// TwinCAT 3 PLC project sample_delivery
// Title: lcsl-plc-icl-sample-delivery
// Company: SLAC
// ProjectVersion: 0.0.0
// ProgramVersion: 3.1.4023.0
// libraries:
//   lcls-twincat-sample-delivery, * (SLAC)
//   Tc2_Standard, * (Beckhoff Automation GmbH)
//   Tc2_System, * (Beckhoff Automation GmbH)
//   Tc3_Module, * (Beckhoff Automation GmbH)
// project tree:
//   GVLs/ GVL_SDS.TcGVL
//   / PlcTask.TcTTO (not stored), SerialComm.TcTTO (not stored)
//   POUs/ MAIN.TcPOU, SerialTxRx.TcPOU (not stored)
// real-time tasks:
//   TASK PlcTask: cycle T#10ms, priority 20, ADS port 351
//   TASK SerialComm: cycle T#5ms, priority 1, ADS port 350
// I/O:
//   DEVICE MAIN (EtherCAT), AmsNetId 0.0.0.0.2.1
//     Term 65 (EK1200) [EK1200-5000 EtherCAT Power supply (2A E-Bus)]
//       Term 66 (EL6070) [EL6070 1Ch. Licensing-Terminal]
//       Term 67 (EK1110) [EK1110 EtherCAT extension]
//     Box 68 (EP9128-0021) [EP9128-0021 8x EtherCAT junction]
//       Term 69 (EP9128-1021) [EP9128-1021 8x EtherCAT junction - Dev A]
//       Term 70 (EP9128-2021) [EP9128-2021 8x EtherCAT junction - Dev B]
//     Box 23 (EP9128-0021) [EP9128-0021 8x EtherCAT junction]
//       Term 71 (EP9128-1021) [EP9128-1021 8x EtherCAT junction - Dev A]
//       Term 72 (EP9128-2021) [EP9128-2021 8x EtherCAT junction - Dev B]
//     ALI (EP1111) [EP1111-0000 ID-Switch]
//     ALI_X (EP7041-0002) [EP7041-0002 1Ch. Stepper motor output stage (50V, 5A)]
//     ALI_Y (EP7041-0002) [EP7041-0002 1Ch. Stepper motor output stage (50V, 5A)]
//     ALI_Z (EP7041-0002) [EP7041-0002 1Ch. Stepper motor output stage (50V, 5A)]
//     ALI_X_ENC (EP5101-0011) [EP5101-0011 1Ch. Inc. Encoder 5V, D-SUB15]
//     ALI_Gauges (EP3174-0002) [EP3174-0002 4Ch. Ana. Input +/-10V, 0-10V, 0/4-20mA configurable]
//     ALI_PropValve (EP7041-0002) [EP7041-0002 1Ch. Stepper motor output stage (50V, 5A)]
//     ALI_Y_ENC (EP5101-0011) [EP5101-0011 1Ch. Inc. Encoder 5V, D-SUB15]
//     ALI_DIO (EP2338-0001) [EP2338-0001 8 Ch. Dig. Input/Output 24V, 0,5A, M8]
//     M3 Selector A (EP1111) [EP1111-0000 ID-Switch]
//     M3 Selector A Digital IO (EP2338-1001) [EP2338-1001 8 Ch. Dig. Input/Output 24V, 3ms, 0,5A, M8]
//     M3 Selector A Serial IO (EP6002-0002) [EP6002-0002 Interface (RS232/422/485)]
//     M3 Selector B (EP1111) [EP1111-0000 ID-Switch]
//     M3 Selector B Digital IO (EP2338-1001) [EP2338-1001 8 Ch. Dig. Input/Output 24V, 3ms, 0,5A, M8]
//     M3 Selector B Serial IO (EP6002-0002) [EP6002-0002 Interface (RS232/422/485)]
//     PCM A (EP1111) [EP1111-0000 ID-Switch]
//     PCM A (EP4374-0002) [EP4374-0002 2Ch. Ana. Input +/-10V, 0-10V, 0/4-20mA configurable; 2Ch. Ana. Output +/-10V, 0-10V, 0/4-20mA configurable]
//     PCM A (EP3174-0002) [EP3174-0002 4Ch. Ana. Input +/-10V, 0-10V, 0/4-20mA configurable]
//     PCM A (EP6002-0002) [EP6002-0002 Interface (RS232/422/485)]
//     PCM B (EP1111) [EP1111-0000 ID-Switch]
//     PCM B (EP4374-0002) [EP4374-0002 2Ch. Ana. Input +/-10V, 0-10V, 0/4-20mA configurable; 2Ch. Ana. Output +/-10V, 0-10V, 0/4-20mA configurable]
//     PCM B (EP3174-0002) [EP3174-0002 4Ch. Ana. Input +/-10V, 0-10V, 0/4-20mA configurable]
//     PCM B (EP6002-0002) [EP6002-0002 Interface (RS232/422/485)]
//     Gas_Mani (EP1111) [EP1111-0000 ID-Switch]
//     Gas_Mani_NeedleValve (EP4374-0002) [EP4374-0002 2Ch. Ana. Input +/-10V, 0-10V, 0/4-20mA configurable; 2Ch. Ana. Output +/-10V, 0-10V, 0/4-20mA configurable]
//     Gas_Mani_ValveCtrl (EP2338-0001) [EP2338-0001 8 Ch. Dig. Input/Output 24V, 0,5A, M8]
//     Gas_Mani_ValveRbk (EP2338-0001) [EP2338-0001 8 Ch. Dig. Input/Output 24V, 0,5A, M8]
//     M3 Selector C (EP1111) [EP1111-0000 ID-Switch]
//     M3 Selector C Digital IO (EP2338-1001) [EP2338-1001 8 Ch. Dig. Input/Output 24V, 3ms, 0,5A, M8]
//     M3 Selector C Serial IO (EP6002-0002) [EP6002-0002 Interface (RS232/422/485)]
//     M3 Selector D (EP1111) [EP1111-0000 ID-Switch]
//     M3 Selector D Digital IO (EP2338-1001) [EP2338-1001 8 Ch. Dig. Input/Output 24V, 3ms, 0,5A, M8]
//     M3 Selector D Serial IO (EP6002-0002) [EP6002-0002 Interface (RS232/422/485)]
//     PCM C (EP1111) [EP1111-0000 ID-Switch]
//     PCM C (EP4374-0002) [EP4374-0002 2Ch. Ana. Input +/-10V, 0-10V, 0/4-20mA configurable; 2Ch. Ana. Output +/-10V, 0-10V, 0/4-20mA configurable]
//     PCM C (EP3174-0002) [EP3174-0002 4Ch. Ana. Input +/-10V, 0-10V, 0/4-20mA configurable]
//     PCM C (EP6002-0002) [EP6002-0002 Interface (RS232/422/485)]
//     PCM D (EP1111) [EP1111-0000 ID-Switch]
//     PCM D (EP4374-0002) [EP4374-0002 2Ch. Ana. Input +/-10V, 0-10V, 0/4-20mA configurable; 2Ch. Ana. Output +/-10V, 0-10V, 0/4-20mA configurable]
//     PCM D (EP3174-0002) [EP3174-0002 4Ch. Ana. Input +/-10V, 0-10V, 0/4-20mA configurable]
//     PCM D (EP6002-0002) [EP6002-0002 Interface (RS232/422/485)]
//     Bronkhorst MFM A [Mass Flow / Pressure Controller - Slave]
//     Bronkhorst MFM B [Mass Flow / Pressure Controller - Slave]
//     Bronkhorst MFM C [Mass Flow / Pressure Controller - Slave]
//     Bronkhorst MFM D [Mass Flow / Pressure Controller - Slave]
//     Solenoid Pair A (EP1111)
//     Solenoid Pair A Digital IO (EP2338-0001)
//     SC5 [EP9128-0021 8x EtherCAT junction]
//       Box 26 (EP9128-1021) [EP9128-1021 8x EtherCAT junction - Dev A]
//       Box 27 (EP9128-2021) [EP9128-2021 8x EtherCAT junction - Dev B]
//     SC4 [EP9128-0021 8x EtherCAT junction]
//       Box 24 (EP9128-1021) [EP9128-1021 8x EtherCAT junction - Dev A]
//       Box 25 (EP9128-2021) [EP9128-2021 8x EtherCAT junction - Dev B]
// variable links:
//   sample_delivery Instance <-> MAIN (EtherCAT)/Bronkhorst MFM A
//     PlcTask Inputs/GVL_SDS.BronkhorstA.stMFM.i_rFlow <-> TxPDO Map/fMeasure
//     PlcTask Outputs/GVL_SDS.BronkhorstA.stMFM.q_rSetpoint <-> RxPDO Map/fSetpoint
//   sample_delivery Instance <-> MAIN (EtherCAT)/Bronkhorst MFM B
//     PlcTask Inputs/GVL_SDS.BronkhorstB.stMFM.i_rFlow <-> TxPDO Map/fMeasure
//     PlcTask Outputs/GVL_SDS.BronkhorstB.stMFM.q_rSetpoint <-> RxPDO Map/fSetpoint
//   sample_delivery Instance <-> MAIN (EtherCAT)/Bronkhorst MFM C
//     PlcTask Inputs/GVL_SDS.BronkhorstC.stMFM.i_rFlow <-> TxPDO Map/fMeasure
//     PlcTask Outputs/GVL_SDS.BronkhorstC.stMFM.q_rSetpoint <-> RxPDO Map/fSetpoint
//   sample_delivery Instance <-> MAIN (EtherCAT)/Bronkhorst MFM D
//     PlcTask Inputs/GVL_SDS.BronkhorstD.stMFM.i_rFlow <-> TxPDO Map/fMeasure
//     PlcTask Outputs/GVL_SDS.BronkhorstD.stMFM.q_rSetpoint <-> RxPDO Map/fSetpoint
//   sample_delivery Instance <-> MAIN (EtherCAT)/Gas_Mani (EP1111)
//     PlcTask Inputs/GVL_SDS.GasMan.stBaseIO.i_SyncUnitWC <-> WcState/WcState
//   sample_delivery Instance <-> MAIN (EtherCAT)/Gas_Mani_ValveCtrl (EP2338-0001)
//     PlcTask Outputs/GVL_SDS.GasMan.stValve[{1..7}].qxDO <-> Channel {9..15}/Output  (7 links)
//   sample_delivery Instance <-> MAIN (EtherCAT)/Gas_Mani_ValveRbk (EP2338-0001)
//     PlcTask Inputs/GVL_SDS.GasMan.stValve[{1..7}].ixOPN <-> Channel {1..7}/Input  (7 links)
//   sample_delivery Instance <-> MAIN (EtherCAT)/M3 Selector A (EP1111)
//     PlcTask Inputs/GVL_SDS.M3SelectorA.stBaseIO.i_SyncUnitWC <-> WcState/WcState
//   sample_delivery Instance <-> MAIN (EtherCAT)/M3 Selector A Digital IO (EP2338-1001)
//     PlcTask Outputs/GVL_SDS.M3SelectorA.stShaker01.q_xPwrDO <-> Channel 9/Output
//     PlcTask Outputs/GVL_SDS.M3SelectorA.stShaker02.q_xPwrDO <-> Channel 10/Output
//     PlcTask Outputs/GVL_SDS.M3SelectorA.stShaker03.q_xPwrDO <-> Channel 11/Output
//     PlcTask Outputs/GVL_SDS.M3SelectorA.stShaker04.q_xPwrDO <-> Channel 12/Output
//   sample_delivery Instance <-> MAIN (EtherCAT)/M3 Selector A Serial IO (EP6002-0002)
//     SerialComm Inputs/GVL_SDS.M3SelectorA.stSensSerial.stComIn/D <-> COM TxPDO-Map Inputs Channel 1/Data In 0
//     SerialComm Inputs/GVL_SDS.M3SelectorA.stSensSerial.stComIn/D @bit {8..168 step 8} <-> COM TxPDO-Map Inputs Channel 1/Data In {1..21}  (21 links)
//     SerialComm Inputs/GVL_SDS.M3SelectorA.stSensSerial.stComIn/Status <-> COM TxPDO-Map Inputs Channel 1/Status
//     SerialComm Inputs/GVL_SDS.M3SelectorA.stViciSerial.stComIn/D <-> COM TxPDO-Map Inputs Channel 2/Data In 0
//     SerialComm Inputs/GVL_SDS.M3SelectorA.stViciSerial.stComIn/D @bit {8..168 step 8} <-> COM TxPDO-Map Inputs Channel 2/Data In {1..21}  (21 links)
//     SerialComm Inputs/GVL_SDS.M3SelectorA.stViciSerial.stComIn/Status <-> COM TxPDO-Map Inputs Channel 2/Status
//     SerialComm Outputs/GVL_SDS.M3SelectorA.stSensSerial.stComOut/Ctrl <-> COM RxPDO-Map Outputs Channel 1/Ctrl
//     SerialComm Outputs/GVL_SDS.M3SelectorA.stSensSerial.stComOut/D <-> COM RxPDO-Map Outputs Channel 1/Data Out 0
//     SerialComm Outputs/GVL_SDS.M3SelectorA.stSensSerial.stComOut/D @bit {8..168 step 8} <-> COM RxPDO-Map Outputs Channel 1/Data Out {1..21}  (21 links)
//     SerialComm Outputs/GVL_SDS.M3SelectorA.stViciSerial.stComOut/Ctrl <-> COM RxPDO-Map Outputs Channel 2/Ctrl
//     SerialComm Outputs/GVL_SDS.M3SelectorA.stViciSerial.stComOut/D <-> COM RxPDO-Map Outputs Channel 2/Data Out 0
//     SerialComm Outputs/GVL_SDS.M3SelectorA.stViciSerial.stComOut/D @bit {8..168 step 8} <-> COM RxPDO-Map Outputs Channel 2/Data Out {1..21}  (21 links)
//   sample_delivery Instance <-> MAIN (EtherCAT)/M3 Selector B (EP1111)
//     PlcTask Inputs/GVL_SDS.M3SelectorB.stBaseIO.i_SyncUnitWC <-> WcState/WcState
//   sample_delivery Instance <-> MAIN (EtherCAT)/M3 Selector B Digital IO (EP2338-1001)
//     PlcTask Outputs/GVL_SDS.M3SelectorB.stShaker01.q_xPwrDO <-> Channel 9/Output
//     PlcTask Outputs/GVL_SDS.M3SelectorB.stShaker02.q_xPwrDO <-> Channel 10/Output
//     PlcTask Outputs/GVL_SDS.M3SelectorB.stShaker03.q_xPwrDO <-> Channel 11/Output
//     PlcTask Outputs/GVL_SDS.M3SelectorB.stShaker04.q_xPwrDO <-> Channel 12/Output
//   sample_delivery Instance <-> MAIN (EtherCAT)/M3 Selector B Serial IO (EP6002-0002)
//     SerialComm Inputs/GVL_SDS.M3SelectorB.stSensSerial.stComIn/D <-> COM TxPDO-Map Inputs Channel 1/Data In 0
//     SerialComm Inputs/GVL_SDS.M3SelectorB.stSensSerial.stComIn/D @bit {8..168 step 8} <-> COM TxPDO-Map Inputs Channel 1/Data In {1..21}  (21 links)
//     SerialComm Inputs/GVL_SDS.M3SelectorB.stSensSerial.stComIn/Status <-> COM TxPDO-Map Inputs Channel 1/Status
//     SerialComm Inputs/GVL_SDS.M3SelectorB.stViciSerial.stComIn/D <-> COM TxPDO-Map Inputs Channel 2/Data In 0
//     SerialComm Inputs/GVL_SDS.M3SelectorB.stViciSerial.stComIn/D @bit {8..168 step 8} <-> COM TxPDO-Map Inputs Channel 2/Data In {1..21}  (21 links)
//     SerialComm Inputs/GVL_SDS.M3SelectorB.stViciSerial.stComIn/Status <-> COM TxPDO-Map Inputs Channel 2/Status
//     SerialComm Outputs/GVL_SDS.M3SelectorB.stSensSerial.stComOut/Ctrl <-> COM RxPDO-Map Outputs Channel 1/Ctrl
//     SerialComm Outputs/GVL_SDS.M3SelectorB.stSensSerial.stComOut/D <-> COM RxPDO-Map Outputs Channel 1/Data Out 0
//     SerialComm Outputs/GVL_SDS.M3SelectorB.stSensSerial.stComOut/D @bit {8..168 step 8} <-> COM RxPDO-Map Outputs Channel 1/Data Out {1..21}  (21 links)
//     SerialComm Outputs/GVL_SDS.M3SelectorB.stViciSerial.stComOut/Ctrl <-> COM RxPDO-Map Outputs Channel 2/Ctrl
//     SerialComm Outputs/GVL_SDS.M3SelectorB.stViciSerial.stComOut/D <-> COM RxPDO-Map Outputs Channel 2/Data Out 0
//     SerialComm Outputs/GVL_SDS.M3SelectorB.stViciSerial.stComOut/D @bit {8..168 step 8} <-> COM RxPDO-Map Outputs Channel 2/Data Out {1..21}  (21 links)
//   sample_delivery Instance <-> MAIN (EtherCAT)/M3 Selector C (EP1111)
//     PlcTask Inputs/GVL_SDS.M3SelectorC.stBaseIO.i_SyncUnitWC <-> WcState/WcState
//   sample_delivery Instance <-> MAIN (EtherCAT)/M3 Selector C Digital IO (EP2338-1001)
//     PlcTask Outputs/GVL_SDS.M3SelectorC.stShaker01.q_xPwrDO <-> Channel 9/Output
//     PlcTask Outputs/GVL_SDS.M3SelectorC.stShaker02.q_xPwrDO <-> Channel 10/Output
//     PlcTask Outputs/GVL_SDS.M3SelectorC.stShaker03.q_xPwrDO <-> Channel 11/Output
//     PlcTask Outputs/GVL_SDS.M3SelectorC.stShaker04.q_xPwrDO <-> Channel 12/Output
//   sample_delivery Instance <-> MAIN (EtherCAT)/M3 Selector C Serial IO (EP6002-0002)
//     SerialComm Inputs/GVL_SDS.M3SelectorC.stSensSerial.stComIn/D <-> COM TxPDO-Map Inputs Channel 1/Data In 0
//     SerialComm Inputs/GVL_SDS.M3SelectorC.stSensSerial.stComIn/D @bit {8..168 step 8} <-> COM TxPDO-Map Inputs Channel 1/Data In {1..21}  (21 links)
//     SerialComm Inputs/GVL_SDS.M3SelectorC.stSensSerial.stComIn/Status <-> COM TxPDO-Map Inputs Channel 1/Status
//     SerialComm Inputs/GVL_SDS.M3SelectorC.stViciSerial.stComIn/D <-> COM TxPDO-Map Inputs Channel 2/Data In 0
//     SerialComm Inputs/GVL_SDS.M3SelectorC.stViciSerial.stComIn/D @bit {8..168 step 8} <-> COM TxPDO-Map Inputs Channel 2/Data In {1..21}  (21 links)
//     SerialComm Inputs/GVL_SDS.M3SelectorC.stViciSerial.stComIn/Status <-> COM TxPDO-Map Inputs Channel 2/Status
//     SerialComm Outputs/GVL_SDS.M3SelectorC.stSensSerial.stComOut/Ctrl <-> COM RxPDO-Map Outputs Channel 1/Ctrl
//     SerialComm Outputs/GVL_SDS.M3SelectorC.stSensSerial.stComOut/D <-> COM RxPDO-Map Outputs Channel 1/Data Out 0
//     SerialComm Outputs/GVL_SDS.M3SelectorC.stSensSerial.stComOut/D @bit {8..168 step 8} <-> COM RxPDO-Map Outputs Channel 1/Data Out {1..21}  (21 links)
//     SerialComm Outputs/GVL_SDS.M3SelectorC.stViciSerial.stComOut/Ctrl <-> COM RxPDO-Map Outputs Channel 2/Ctrl
//     SerialComm Outputs/GVL_SDS.M3SelectorC.stViciSerial.stComOut/D <-> COM RxPDO-Map Outputs Channel 2/Data Out 0
//     SerialComm Outputs/GVL_SDS.M3SelectorC.stViciSerial.stComOut/D @bit {8..168 step 8} <-> COM RxPDO-Map Outputs Channel 2/Data Out {1..21}  (21 links)
//   sample_delivery Instance <-> MAIN (EtherCAT)/M3 Selector D (EP1111)
//     PlcTask Inputs/GVL_SDS.M3SelectorD.stBaseIO.i_SyncUnitWC <-> WcState/WcState
//   sample_delivery Instance <-> MAIN (EtherCAT)/M3 Selector D Digital IO (EP2338-1001)
//     PlcTask Outputs/GVL_SDS.M3SelectorD.stShaker01.q_xPwrDO <-> Channel 9/Output
//     PlcTask Outputs/GVL_SDS.M3SelectorD.stShaker02.q_xPwrDO <-> Channel 10/Output
//     PlcTask Outputs/GVL_SDS.M3SelectorD.stShaker03.q_xPwrDO <-> Channel 11/Output
//     PlcTask Outputs/GVL_SDS.M3SelectorD.stShaker04.q_xPwrDO <-> Channel 12/Output
//   sample_delivery Instance <-> MAIN (EtherCAT)/M3 Selector D Serial IO (EP6002-0002)
//     SerialComm Inputs/GVL_SDS.M3SelectorD.stSensSerial.stComIn/D <-> COM TxPDO-Map Inputs Channel 1/Data In 0
//     SerialComm Inputs/GVL_SDS.M3SelectorD.stSensSerial.stComIn/D @bit {8..168 step 8} <-> COM TxPDO-Map Inputs Channel 1/Data In {1..21}  (21 links)
//     SerialComm Inputs/GVL_SDS.M3SelectorD.stSensSerial.stComIn/Status <-> COM TxPDO-Map Inputs Channel 1/Status
//     SerialComm Inputs/GVL_SDS.M3SelectorD.stViciSerial.stComIn/D <-> COM TxPDO-Map Inputs Channel 2/Data In 0
//     SerialComm Inputs/GVL_SDS.M3SelectorD.stViciSerial.stComIn/D @bit {8..168 step 8} <-> COM TxPDO-Map Inputs Channel 2/Data In {1..21}  (21 links)
//     SerialComm Inputs/GVL_SDS.M3SelectorD.stViciSerial.stComIn/Status <-> COM TxPDO-Map Inputs Channel 2/Status
//     SerialComm Outputs/GVL_SDS.M3SelectorD.stSensSerial.stComOut/Ctrl <-> COM RxPDO-Map Outputs Channel 1/Ctrl
//     SerialComm Outputs/GVL_SDS.M3SelectorD.stSensSerial.stComOut/D <-> COM RxPDO-Map Outputs Channel 1/Data Out 0
//     SerialComm Outputs/GVL_SDS.M3SelectorD.stSensSerial.stComOut/D @bit {8..168 step 8} <-> COM RxPDO-Map Outputs Channel 1/Data Out {1..21}  (21 links)
//     SerialComm Outputs/GVL_SDS.M3SelectorD.stViciSerial.stComOut/Ctrl <-> COM RxPDO-Map Outputs Channel 2/Ctrl
//     SerialComm Outputs/GVL_SDS.M3SelectorD.stViciSerial.stComOut/D <-> COM RxPDO-Map Outputs Channel 2/Data Out 0
//     SerialComm Outputs/GVL_SDS.M3SelectorD.stViciSerial.stComOut/D @bit {8..168 step 8} <-> COM RxPDO-Map Outputs Channel 2/Data Out {1..21}  (21 links)
//   sample_delivery Instance <-> MAIN (EtherCAT)/PCM A (EP1111)
//     PlcTask Inputs/GVL_SDS.PCMA.stBaseIO.i_SyncUnitWC <-> WcState/WcState
//   sample_delivery Instance <-> MAIN (EtherCAT)/PCM A (EP4374-0002)
//     PlcTask Inputs/GVL_SDS.PCMA.stPropAir1.i_iPressRB <-> AI Inputs Channel 1/Value
//     PlcTask Inputs/GVL_SDS.PCMA.stPropAir2.i_iPressRB <-> AI Inputs Channel 2/Value
//     PlcTask Outputs/GVL_SDS.PCMA.stPropAir1.q_iPressCt <-> AO Outputs Channel 3/Analog output
//     PlcTask Outputs/GVL_SDS.PCMA.stPropAir2.q_iPressCt <-> AO Outputs Channel 4/Analog output
//   sample_delivery Instance <-> MAIN (EtherCAT)/PCM A (EP6002-0002)
//     SerialComm Inputs/GVL_SDS.PCMA.stSerial1.stComIn/D <-> COM TxPDO-Map Inputs Channel 1/Data In 0
//     SerialComm Inputs/GVL_SDS.PCMA.stSerial2.stComIn/D <-> COM TxPDO-Map Inputs Channel 2/Data In 0
//     SerialComm Inputs/GVL_SDS.PCMA.stSerial1.stComIn/D @bit 8 <-> COM TxPDO-Map Inputs Channel 1/Data In 1
//     SerialComm Inputs/GVL_SDS.PCMA.stSerial1.stComIn/D @bit 80 <-> COM TxPDO-Map Inputs Channel 1/Data In 10
//     SerialComm Inputs/GVL_SDS.PCMA.stSerial1.stComIn/D @bit 88 <-> COM TxPDO-Map Inputs Channel 1/Data In 11
//     SerialComm Inputs/GVL_SDS.PCMA.stSerial1.stComIn/D @bit 96 <-> COM TxPDO-Map Inputs Channel 1/Data In 12
//     SerialComm Inputs/GVL_SDS.PCMA.stSerial1.stComIn/D @bit 104 <-> COM TxPDO-Map Inputs Channel 1/Data In 13
//     SerialComm Inputs/GVL_SDS.PCMA.stSerial1.stComIn/D @bit 112 <-> COM TxPDO-Map Inputs Channel 1/Data In 14
//     SerialComm Inputs/GVL_SDS.PCMA.stSerial1.stComIn/D @bit 120 <-> COM TxPDO-Map Inputs Channel 1/Data In 15
//     SerialComm Inputs/GVL_SDS.PCMA.stSerial1.stComIn/D @bit 128 <-> COM TxPDO-Map Inputs Channel 1/Data In 16
//     SerialComm Inputs/GVL_SDS.PCMA.stSerial1.stComIn/D @bit 136 <-> COM TxPDO-Map Inputs Channel 1/Data In 17
//     SerialComm Inputs/GVL_SDS.PCMA.stSerial1.stComIn/D @bit 144 <-> COM TxPDO-Map Inputs Channel 1/Data In 18
//     SerialComm Inputs/GVL_SDS.PCMA.stSerial1.stComIn/D @bit 152 <-> COM TxPDO-Map Inputs Channel 1/Data In 19
//     SerialComm Inputs/GVL_SDS.PCMA.stSerial1.stComIn/D @bit 16 <-> COM TxPDO-Map Inputs Channel 1/Data In 2
//     SerialComm Inputs/GVL_SDS.PCMA.stSerial1.stComIn/D @bit 160 <-> COM TxPDO-Map Inputs Channel 1/Data In 20
//     SerialComm Inputs/GVL_SDS.PCMA.stSerial1.stComIn/D @bit 168 <-> COM TxPDO-Map Inputs Channel 1/Data In 21
//     SerialComm Inputs/GVL_SDS.PCMA.stSerial1.stComIn/D @bit 24 <-> COM TxPDO-Map Inputs Channel 1/Data In 3
//     SerialComm Inputs/GVL_SDS.PCMA.stSerial1.stComIn/D @bit 32 <-> COM TxPDO-Map Inputs Channel 1/Data In 4
//     SerialComm Inputs/GVL_SDS.PCMA.stSerial1.stComIn/D @bit 40 <-> COM TxPDO-Map Inputs Channel 1/Data In 5
//     SerialComm Inputs/GVL_SDS.PCMA.stSerial1.stComIn/D @bit 48 <-> COM TxPDO-Map Inputs Channel 1/Data In 6
//     SerialComm Inputs/GVL_SDS.PCMA.stSerial1.stComIn/D @bit 56 <-> COM TxPDO-Map Inputs Channel 1/Data In 7
//     SerialComm Inputs/GVL_SDS.PCMA.stSerial1.stComIn/D @bit 64 <-> COM TxPDO-Map Inputs Channel 1/Data In 8
//     SerialComm Inputs/GVL_SDS.PCMA.stSerial1.stComIn/D @bit 72 <-> COM TxPDO-Map Inputs Channel 1/Data In 9
//     SerialComm Inputs/GVL_SDS.PCMA.stSerial2.stComIn/D @bit 8 <-> COM TxPDO-Map Inputs Channel 2/Data In 1
//     SerialComm Inputs/GVL_SDS.PCMA.stSerial2.stComIn/D @bit 80 <-> COM TxPDO-Map Inputs Channel 2/Data In 10
//     SerialComm Inputs/GVL_SDS.PCMA.stSerial2.stComIn/D @bit 88 <-> COM TxPDO-Map Inputs Channel 2/Data In 11
//     SerialComm Inputs/GVL_SDS.PCMA.stSerial2.stComIn/D @bit 96 <-> COM TxPDO-Map Inputs Channel 2/Data In 12
//     SerialComm Inputs/GVL_SDS.PCMA.stSerial2.stComIn/D @bit 104 <-> COM TxPDO-Map Inputs Channel 2/Data In 13
//     SerialComm Inputs/GVL_SDS.PCMA.stSerial2.stComIn/D @bit 112 <-> COM TxPDO-Map Inputs Channel 2/Data In 14
//     SerialComm Inputs/GVL_SDS.PCMA.stSerial2.stComIn/D @bit 120 <-> COM TxPDO-Map Inputs Channel 2/Data In 15
//     SerialComm Inputs/GVL_SDS.PCMA.stSerial2.stComIn/D @bit 128 <-> COM TxPDO-Map Inputs Channel 2/Data In 16
//     SerialComm Inputs/GVL_SDS.PCMA.stSerial2.stComIn/D @bit 136 <-> COM TxPDO-Map Inputs Channel 2/Data In 17
//     SerialComm Inputs/GVL_SDS.PCMA.stSerial2.stComIn/D @bit 144 <-> COM TxPDO-Map Inputs Channel 2/Data In 18
//     SerialComm Inputs/GVL_SDS.PCMA.stSerial2.stComIn/D @bit 152 <-> COM TxPDO-Map Inputs Channel 2/Data In 19
//     SerialComm Inputs/GVL_SDS.PCMA.stSerial2.stComIn/D @bit 16 <-> COM TxPDO-Map Inputs Channel 2/Data In 2
//     SerialComm Inputs/GVL_SDS.PCMA.stSerial2.stComIn/D @bit 160 <-> COM TxPDO-Map Inputs Channel 2/Data In 20
//     SerialComm Inputs/GVL_SDS.PCMA.stSerial2.stComIn/D @bit 168 <-> COM TxPDO-Map Inputs Channel 2/Data In 21
//     SerialComm Inputs/GVL_SDS.PCMA.stSerial2.stComIn/D @bit 24 <-> COM TxPDO-Map Inputs Channel 2/Data In 3
//     SerialComm Inputs/GVL_SDS.PCMA.stSerial2.stComIn/D @bit 32 <-> COM TxPDO-Map Inputs Channel 2/Data In 4
//     SerialComm Inputs/GVL_SDS.PCMA.stSerial2.stComIn/D @bit 40 <-> COM TxPDO-Map Inputs Channel 2/Data In 5
//     SerialComm Inputs/GVL_SDS.PCMA.stSerial2.stComIn/D @bit 48 <-> COM TxPDO-Map Inputs Channel 2/Data In 6
//     SerialComm Inputs/GVL_SDS.PCMA.stSerial2.stComIn/D @bit 56 <-> COM TxPDO-Map Inputs Channel 2/Data In 7
//     SerialComm Inputs/GVL_SDS.PCMA.stSerial2.stComIn/D @bit 64 <-> COM TxPDO-Map Inputs Channel 2/Data In 8
//     SerialComm Inputs/GVL_SDS.PCMA.stSerial2.stComIn/D @bit 72 <-> COM TxPDO-Map Inputs Channel 2/Data In 9
//     SerialComm Inputs/GVL_SDS.PCMA.stSerial1.stComIn/Status <-> COM TxPDO-Map Inputs Channel 1/Status
//     SerialComm Inputs/GVL_SDS.PCMA.stSerial2.stComIn/Status <-> COM TxPDO-Map Inputs Channel 2/Status
//     SerialComm Outputs/GVL_SDS.PCMA.stSerial1.stComOut/Ctrl <-> COM RxPDO-Map Outputs Channel 1/Ctrl
//     SerialComm Outputs/GVL_SDS.PCMA.stSerial2.stComOut/Ctrl <-> COM RxPDO-Map Outputs Channel 2/Ctrl
//     SerialComm Outputs/GVL_SDS.PCMA.stSerial1.stComOut/D <-> COM RxPDO-Map Outputs Channel 1/Data Out 0
//     SerialComm Outputs/GVL_SDS.PCMA.stSerial2.stComOut/D <-> COM RxPDO-Map Outputs Channel 2/Data Out 0
//     SerialComm Outputs/GVL_SDS.PCMA.stSerial1.stComOut/D @bit 8 <-> COM RxPDO-Map Outputs Channel 1/Data Out 1
//     SerialComm Outputs/GVL_SDS.PCMA.stSerial1.stComOut/D @bit 80 <-> COM RxPDO-Map Outputs Channel 1/Data Out 10
//     SerialComm Outputs/GVL_SDS.PCMA.stSerial1.stComOut/D @bit 88 <-> COM RxPDO-Map Outputs Channel 1/Data Out 11
//     SerialComm Outputs/GVL_SDS.PCMA.stSerial1.stComOut/D @bit 96 <-> COM RxPDO-Map Outputs Channel 1/Data Out 12
//     SerialComm Outputs/GVL_SDS.PCMA.stSerial1.stComOut/D @bit 104 <-> COM RxPDO-Map Outputs Channel 1/Data Out 13
//     SerialComm Outputs/GVL_SDS.PCMA.stSerial1.stComOut/D @bit 112 <-> COM RxPDO-Map Outputs Channel 1/Data Out 14
//     SerialComm Outputs/GVL_SDS.PCMA.stSerial1.stComOut/D @bit 120 <-> COM RxPDO-Map Outputs Channel 1/Data Out 15
//     SerialComm Outputs/GVL_SDS.PCMA.stSerial1.stComOut/D @bit 128 <-> COM RxPDO-Map Outputs Channel 1/Data Out 16
//     SerialComm Outputs/GVL_SDS.PCMA.stSerial1.stComOut/D @bit 136 <-> COM RxPDO-Map Outputs Channel 1/Data Out 17
//     SerialComm Outputs/GVL_SDS.PCMA.stSerial1.stComOut/D @bit 144 <-> COM RxPDO-Map Outputs Channel 1/Data Out 18
//     SerialComm Outputs/GVL_SDS.PCMA.stSerial1.stComOut/D @bit 152 <-> COM RxPDO-Map Outputs Channel 1/Data Out 19
//     SerialComm Outputs/GVL_SDS.PCMA.stSerial1.stComOut/D @bit 16 <-> COM RxPDO-Map Outputs Channel 1/Data Out 2
//     SerialComm Outputs/GVL_SDS.PCMA.stSerial1.stComOut/D @bit 160 <-> COM RxPDO-Map Outputs Channel 1/Data Out 20
//     SerialComm Outputs/GVL_SDS.PCMA.stSerial1.stComOut/D @bit 168 <-> COM RxPDO-Map Outputs Channel 1/Data Out 21
//     SerialComm Outputs/GVL_SDS.PCMA.stSerial1.stComOut/D @bit 24 <-> COM RxPDO-Map Outputs Channel 1/Data Out 3
//     SerialComm Outputs/GVL_SDS.PCMA.stSerial1.stComOut/D @bit 32 <-> COM RxPDO-Map Outputs Channel 1/Data Out 4
//     SerialComm Outputs/GVL_SDS.PCMA.stSerial1.stComOut/D @bit 40 <-> COM RxPDO-Map Outputs Channel 1/Data Out 5
//     SerialComm Outputs/GVL_SDS.PCMA.stSerial1.stComOut/D @bit 48 <-> COM RxPDO-Map Outputs Channel 1/Data Out 6
//     SerialComm Outputs/GVL_SDS.PCMA.stSerial1.stComOut/D @bit 56 <-> COM RxPDO-Map Outputs Channel 1/Data Out 7
//     SerialComm Outputs/GVL_SDS.PCMA.stSerial1.stComOut/D @bit 64 <-> COM RxPDO-Map Outputs Channel 1/Data Out 8
//     SerialComm Outputs/GVL_SDS.PCMA.stSerial1.stComOut/D @bit 72 <-> COM RxPDO-Map Outputs Channel 1/Data Out 9
//     SerialComm Outputs/GVL_SDS.PCMA.stSerial2.stComOut/D @bit 8 <-> COM RxPDO-Map Outputs Channel 2/Data Out 1
//     SerialComm Outputs/GVL_SDS.PCMA.stSerial2.stComOut/D @bit 80 <-> COM RxPDO-Map Outputs Channel 2/Data Out 10
//     SerialComm Outputs/GVL_SDS.PCMA.stSerial2.stComOut/D @bit 88 <-> COM RxPDO-Map Outputs Channel 2/Data Out 11
//     SerialComm Outputs/GVL_SDS.PCMA.stSerial2.stComOut/D @bit 96 <-> COM RxPDO-Map Outputs Channel 2/Data Out 12
//     SerialComm Outputs/GVL_SDS.PCMA.stSerial2.stComOut/D @bit 104 <-> COM RxPDO-Map Outputs Channel 2/Data Out 13
//     SerialComm Outputs/GVL_SDS.PCMA.stSerial2.stComOut/D @bit 112 <-> COM RxPDO-Map Outputs Channel 2/Data Out 14
//     SerialComm Outputs/GVL_SDS.PCMA.stSerial2.stComOut/D @bit 120 <-> COM RxPDO-Map Outputs Channel 2/Data Out 15
//     SerialComm Outputs/GVL_SDS.PCMA.stSerial2.stComOut/D @bit 128 <-> COM RxPDO-Map Outputs Channel 2/Data Out 16
//     SerialComm Outputs/GVL_SDS.PCMA.stSerial2.stComOut/D @bit 136 <-> COM RxPDO-Map Outputs Channel 2/Data Out 17
//     SerialComm Outputs/GVL_SDS.PCMA.stSerial2.stComOut/D @bit 144 <-> COM RxPDO-Map Outputs Channel 2/Data Out 18
//     SerialComm Outputs/GVL_SDS.PCMA.stSerial2.stComOut/D @bit 152 <-> COM RxPDO-Map Outputs Channel 2/Data Out 19
//     SerialComm Outputs/GVL_SDS.PCMA.stSerial2.stComOut/D @bit 16 <-> COM RxPDO-Map Outputs Channel 2/Data Out 2
//     SerialComm Outputs/GVL_SDS.PCMA.stSerial2.stComOut/D @bit 160 <-> COM RxPDO-Map Outputs Channel 2/Data Out 20
//     SerialComm Outputs/GVL_SDS.PCMA.stSerial2.stComOut/D @bit 168 <-> COM RxPDO-Map Outputs Channel 2/Data Out 21
//     SerialComm Outputs/GVL_SDS.PCMA.stSerial2.stComOut/D @bit 24 <-> COM RxPDO-Map Outputs Channel 2/Data Out 3
//     SerialComm Outputs/GVL_SDS.PCMA.stSerial2.stComOut/D @bit 32 <-> COM RxPDO-Map Outputs Channel 2/Data Out 4
//     SerialComm Outputs/GVL_SDS.PCMA.stSerial2.stComOut/D @bit 40 <-> COM RxPDO-Map Outputs Channel 2/Data Out 5
//     SerialComm Outputs/GVL_SDS.PCMA.stSerial2.stComOut/D @bit 48 <-> COM RxPDO-Map Outputs Channel 2/Data Out 6
//     SerialComm Outputs/GVL_SDS.PCMA.stSerial2.stComOut/D @bit 56 <-> COM RxPDO-Map Outputs Channel 2/Data Out 7
//     SerialComm Outputs/GVL_SDS.PCMA.stSerial2.stComOut/D @bit 64 <-> COM RxPDO-Map Outputs Channel 2/Data Out 8
//     SerialComm Outputs/GVL_SDS.PCMA.stSerial2.stComOut/D @bit 72 <-> COM RxPDO-Map Outputs Channel 2/Data Out 9
//   sample_delivery Instance <-> MAIN (EtherCAT)/PCM B (EP1111)
//     PlcTask Inputs/GVL_SDS.PCMB.stBaseIO.i_SyncUnitWC <-> WcState/WcState
//   sample_delivery Instance <-> MAIN (EtherCAT)/PCM B (EP4374-0002)
//     PlcTask Inputs/GVL_SDS.PCMB.stPropAir1.i_iPressRB <-> AI Inputs Channel 1/Value
//     PlcTask Inputs/GVL_SDS.PCMB.stPropAir2.i_iPressRB <-> AI Inputs Channel 2/Value
//     PlcTask Outputs/GVL_SDS.PCMB.stPropAir1.q_iPressCt <-> AO Outputs Channel 3/Analog output
//     PlcTask Outputs/GVL_SDS.PCMB.stPropAir2.q_iPressCt <-> AO Outputs Channel 4/Analog output
//   sample_delivery Instance <-> MAIN (EtherCAT)/PCM B (EP6002-0002)
//     SerialComm Inputs/GVL_SDS.PCMB.stSerial1.stComIn/D <-> COM TxPDO-Map Inputs Channel 1/Data In 0
//     SerialComm Inputs/GVL_SDS.PCMB.stSerial2.stComIn/D <-> COM TxPDO-Map Inputs Channel 2/Data In 0
//     SerialComm Inputs/GVL_SDS.PCMB.stSerial1.stComIn/D @bit 8 <-> COM TxPDO-Map Inputs Channel 1/Data In 1
//     SerialComm Inputs/GVL_SDS.PCMB.stSerial1.stComIn/D @bit 80 <-> COM TxPDO-Map Inputs Channel 1/Data In 10
//     SerialComm Inputs/GVL_SDS.PCMB.stSerial1.stComIn/D @bit 88 <-> COM TxPDO-Map Inputs Channel 1/Data In 11
//     SerialComm Inputs/GVL_SDS.PCMB.stSerial1.stComIn/D @bit 96 <-> COM TxPDO-Map Inputs Channel 1/Data In 12
//     SerialComm Inputs/GVL_SDS.PCMB.stSerial1.stComIn/D @bit 104 <-> COM TxPDO-Map Inputs Channel 1/Data In 13
//     SerialComm Inputs/GVL_SDS.PCMB.stSerial1.stComIn/D @bit 112 <-> COM TxPDO-Map Inputs Channel 1/Data In 14
//     SerialComm Inputs/GVL_SDS.PCMB.stSerial1.stComIn/D @bit 120 <-> COM TxPDO-Map Inputs Channel 1/Data In 15
//     SerialComm Inputs/GVL_SDS.PCMB.stSerial1.stComIn/D @bit 128 <-> COM TxPDO-Map Inputs Channel 1/Data In 16
//     SerialComm Inputs/GVL_SDS.PCMB.stSerial1.stComIn/D @bit 136 <-> COM TxPDO-Map Inputs Channel 1/Data In 17
//     SerialComm Inputs/GVL_SDS.PCMB.stSerial1.stComIn/D @bit 144 <-> COM TxPDO-Map Inputs Channel 1/Data In 18
//     SerialComm Inputs/GVL_SDS.PCMB.stSerial1.stComIn/D @bit 152 <-> COM TxPDO-Map Inputs Channel 1/Data In 19
//     SerialComm Inputs/GVL_SDS.PCMB.stSerial1.stComIn/D @bit 16 <-> COM TxPDO-Map Inputs Channel 1/Data In 2
//     SerialComm Inputs/GVL_SDS.PCMB.stSerial1.stComIn/D @bit 160 <-> COM TxPDO-Map Inputs Channel 1/Data In 20
//     SerialComm Inputs/GVL_SDS.PCMB.stSerial1.stComIn/D @bit 168 <-> COM TxPDO-Map Inputs Channel 1/Data In 21
//     SerialComm Inputs/GVL_SDS.PCMB.stSerial1.stComIn/D @bit 24 <-> COM TxPDO-Map Inputs Channel 1/Data In 3
//     SerialComm Inputs/GVL_SDS.PCMB.stSerial1.stComIn/D @bit 32 <-> COM TxPDO-Map Inputs Channel 1/Data In 4
//     SerialComm Inputs/GVL_SDS.PCMB.stSerial1.stComIn/D @bit 40 <-> COM TxPDO-Map Inputs Channel 1/Data In 5
//     SerialComm Inputs/GVL_SDS.PCMB.stSerial1.stComIn/D @bit 48 <-> COM TxPDO-Map Inputs Channel 1/Data In 6
//     SerialComm Inputs/GVL_SDS.PCMB.stSerial1.stComIn/D @bit 56 <-> COM TxPDO-Map Inputs Channel 1/Data In 7
//     SerialComm Inputs/GVL_SDS.PCMB.stSerial1.stComIn/D @bit 64 <-> COM TxPDO-Map Inputs Channel 1/Data In 8
//     SerialComm Inputs/GVL_SDS.PCMB.stSerial1.stComIn/D @bit 72 <-> COM TxPDO-Map Inputs Channel 1/Data In 9
//     SerialComm Inputs/GVL_SDS.PCMB.stSerial2.stComIn/D @bit 8 <-> COM TxPDO-Map Inputs Channel 2/Data In 1
//     SerialComm Inputs/GVL_SDS.PCMB.stSerial2.stComIn/D @bit 80 <-> COM TxPDO-Map Inputs Channel 2/Data In 10
//     SerialComm Inputs/GVL_SDS.PCMB.stSerial2.stComIn/D @bit 88 <-> COM TxPDO-Map Inputs Channel 2/Data In 11
//     SerialComm Inputs/GVL_SDS.PCMB.stSerial2.stComIn/D @bit 96 <-> COM TxPDO-Map Inputs Channel 2/Data In 12
//     SerialComm Inputs/GVL_SDS.PCMB.stSerial2.stComIn/D @bit 104 <-> COM TxPDO-Map Inputs Channel 2/Data In 13
//     SerialComm Inputs/GVL_SDS.PCMB.stSerial2.stComIn/D @bit 112 <-> COM TxPDO-Map Inputs Channel 2/Data In 14
//     SerialComm Inputs/GVL_SDS.PCMB.stSerial2.stComIn/D @bit 120 <-> COM TxPDO-Map Inputs Channel 2/Data In 15
//     SerialComm Inputs/GVL_SDS.PCMB.stSerial2.stComIn/D @bit 128 <-> COM TxPDO-Map Inputs Channel 2/Data In 16
//     SerialComm Inputs/GVL_SDS.PCMB.stSerial2.stComIn/D @bit 136 <-> COM TxPDO-Map Inputs Channel 2/Data In 17
//     SerialComm Inputs/GVL_SDS.PCMB.stSerial2.stComIn/D @bit 144 <-> COM TxPDO-Map Inputs Channel 2/Data In 18
//     SerialComm Inputs/GVL_SDS.PCMB.stSerial2.stComIn/D @bit 152 <-> COM TxPDO-Map Inputs Channel 2/Data In 19
//     SerialComm Inputs/GVL_SDS.PCMB.stSerial2.stComIn/D @bit 16 <-> COM TxPDO-Map Inputs Channel 2/Data In 2
//     SerialComm Inputs/GVL_SDS.PCMB.stSerial2.stComIn/D @bit 160 <-> COM TxPDO-Map Inputs Channel 2/Data In 20
//     SerialComm Inputs/GVL_SDS.PCMB.stSerial2.stComIn/D @bit 168 <-> COM TxPDO-Map Inputs Channel 2/Data In 21
//     SerialComm Inputs/GVL_SDS.PCMB.stSerial2.stComIn/D @bit 24 <-> COM TxPDO-Map Inputs Channel 2/Data In 3
//     SerialComm Inputs/GVL_SDS.PCMB.stSerial2.stComIn/D @bit 32 <-> COM TxPDO-Map Inputs Channel 2/Data In 4
//     SerialComm Inputs/GVL_SDS.PCMB.stSerial2.stComIn/D @bit 40 <-> COM TxPDO-Map Inputs Channel 2/Data In 5
//     SerialComm Inputs/GVL_SDS.PCMB.stSerial2.stComIn/D @bit 48 <-> COM TxPDO-Map Inputs Channel 2/Data In 6
//     SerialComm Inputs/GVL_SDS.PCMB.stSerial2.stComIn/D @bit 56 <-> COM TxPDO-Map Inputs Channel 2/Data In 7
//     SerialComm Inputs/GVL_SDS.PCMB.stSerial2.stComIn/D @bit 64 <-> COM TxPDO-Map Inputs Channel 2/Data In 8
//     SerialComm Inputs/GVL_SDS.PCMB.stSerial2.stComIn/D @bit 72 <-> COM TxPDO-Map Inputs Channel 2/Data In 9
//     SerialComm Inputs/GVL_SDS.PCMB.stSerial1.stComIn/Status <-> COM TxPDO-Map Inputs Channel 1/Status
//     SerialComm Inputs/GVL_SDS.PCMB.stSerial2.stComIn/Status <-> COM TxPDO-Map Inputs Channel 2/Status
//     SerialComm Outputs/GVL_SDS.PCMB.stSerial1.stComOut/Ctrl <-> COM RxPDO-Map Outputs Channel 1/Ctrl
//     SerialComm Outputs/GVL_SDS.PCMB.stSerial2.stComOut/Ctrl <-> COM RxPDO-Map Outputs Channel 2/Ctrl
//     SerialComm Outputs/GVL_SDS.PCMB.stSerial1.stComOut/D <-> COM RxPDO-Map Outputs Channel 1/Data Out 0
//     SerialComm Outputs/GVL_SDS.PCMB.stSerial2.stComOut/D <-> COM RxPDO-Map Outputs Channel 2/Data Out 0
//     SerialComm Outputs/GVL_SDS.PCMB.stSerial1.stComOut/D @bit 8 <-> COM RxPDO-Map Outputs Channel 1/Data Out 1
//     SerialComm Outputs/GVL_SDS.PCMB.stSerial1.stComOut/D @bit 80 <-> COM RxPDO-Map Outputs Channel 1/Data Out 10
//     SerialComm Outputs/GVL_SDS.PCMB.stSerial1.stComOut/D @bit 88 <-> COM RxPDO-Map Outputs Channel 1/Data Out 11
//     SerialComm Outputs/GVL_SDS.PCMB.stSerial1.stComOut/D @bit 96 <-> COM RxPDO-Map Outputs Channel 1/Data Out 12
//     SerialComm Outputs/GVL_SDS.PCMB.stSerial1.stComOut/D @bit 104 <-> COM RxPDO-Map Outputs Channel 1/Data Out 13
//     SerialComm Outputs/GVL_SDS.PCMB.stSerial1.stComOut/D @bit 112 <-> COM RxPDO-Map Outputs Channel 1/Data Out 14
//     SerialComm Outputs/GVL_SDS.PCMB.stSerial1.stComOut/D @bit 120 <-> COM RxPDO-Map Outputs Channel 1/Data Out 15
//     SerialComm Outputs/GVL_SDS.PCMB.stSerial1.stComOut/D @bit 128 <-> COM RxPDO-Map Outputs Channel 1/Data Out 16
//     SerialComm Outputs/GVL_SDS.PCMB.stSerial1.stComOut/D @bit 136 <-> COM RxPDO-Map Outputs Channel 1/Data Out 17
//     SerialComm Outputs/GVL_SDS.PCMB.stSerial1.stComOut/D @bit 144 <-> COM RxPDO-Map Outputs Channel 1/Data Out 18
//     SerialComm Outputs/GVL_SDS.PCMB.stSerial1.stComOut/D @bit 152 <-> COM RxPDO-Map Outputs Channel 1/Data Out 19
//     SerialComm Outputs/GVL_SDS.PCMB.stSerial1.stComOut/D @bit 16 <-> COM RxPDO-Map Outputs Channel 1/Data Out 2
//     SerialComm Outputs/GVL_SDS.PCMB.stSerial1.stComOut/D @bit 160 <-> COM RxPDO-Map Outputs Channel 1/Data Out 20
//     SerialComm Outputs/GVL_SDS.PCMB.stSerial1.stComOut/D @bit 168 <-> COM RxPDO-Map Outputs Channel 1/Data Out 21
//     SerialComm Outputs/GVL_SDS.PCMB.stSerial1.stComOut/D @bit 24 <-> COM RxPDO-Map Outputs Channel 1/Data Out 3
//     SerialComm Outputs/GVL_SDS.PCMB.stSerial1.stComOut/D @bit 32 <-> COM RxPDO-Map Outputs Channel 1/Data Out 4
//     SerialComm Outputs/GVL_SDS.PCMB.stSerial1.stComOut/D @bit 40 <-> COM RxPDO-Map Outputs Channel 1/Data Out 5
//     SerialComm Outputs/GVL_SDS.PCMB.stSerial1.stComOut/D @bit 48 <-> COM RxPDO-Map Outputs Channel 1/Data Out 6
//     SerialComm Outputs/GVL_SDS.PCMB.stSerial1.stComOut/D @bit 56 <-> COM RxPDO-Map Outputs Channel 1/Data Out 7
//     SerialComm Outputs/GVL_SDS.PCMB.stSerial1.stComOut/D @bit 64 <-> COM RxPDO-Map Outputs Channel 1/Data Out 8
//     SerialComm Outputs/GVL_SDS.PCMB.stSerial1.stComOut/D @bit 72 <-> COM RxPDO-Map Outputs Channel 1/Data Out 9
//     SerialComm Outputs/GVL_SDS.PCMB.stSerial2.stComOut/D @bit 8 <-> COM RxPDO-Map Outputs Channel 2/Data Out 1
//     SerialComm Outputs/GVL_SDS.PCMB.stSerial2.stComOut/D @bit 80 <-> COM RxPDO-Map Outputs Channel 2/Data Out 10
//     SerialComm Outputs/GVL_SDS.PCMB.stSerial2.stComOut/D @bit 88 <-> COM RxPDO-Map Outputs Channel 2/Data Out 11
//     SerialComm Outputs/GVL_SDS.PCMB.stSerial2.stComOut/D @bit 96 <-> COM RxPDO-Map Outputs Channel 2/Data Out 12
//     SerialComm Outputs/GVL_SDS.PCMB.stSerial2.stComOut/D @bit 104 <-> COM RxPDO-Map Outputs Channel 2/Data Out 13
//     SerialComm Outputs/GVL_SDS.PCMB.stSerial2.stComOut/D @bit 112 <-> COM RxPDO-Map Outputs Channel 2/Data Out 14
//     SerialComm Outputs/GVL_SDS.PCMB.stSerial2.stComOut/D @bit 120 <-> COM RxPDO-Map Outputs Channel 2/Data Out 15
//     SerialComm Outputs/GVL_SDS.PCMB.stSerial2.stComOut/D @bit 128 <-> COM RxPDO-Map Outputs Channel 2/Data Out 16
//     SerialComm Outputs/GVL_SDS.PCMB.stSerial2.stComOut/D @bit 136 <-> COM RxPDO-Map Outputs Channel 2/Data Out 17
//     SerialComm Outputs/GVL_SDS.PCMB.stSerial2.stComOut/D @bit 144 <-> COM RxPDO-Map Outputs Channel 2/Data Out 18
//     SerialComm Outputs/GVL_SDS.PCMB.stSerial2.stComOut/D @bit 152 <-> COM RxPDO-Map Outputs Channel 2/Data Out 19
//     SerialComm Outputs/GVL_SDS.PCMB.stSerial2.stComOut/D @bit 16 <-> COM RxPDO-Map Outputs Channel 2/Data Out 2
//     SerialComm Outputs/GVL_SDS.PCMB.stSerial2.stComOut/D @bit 160 <-> COM RxPDO-Map Outputs Channel 2/Data Out 20
//     SerialComm Outputs/GVL_SDS.PCMB.stSerial2.stComOut/D @bit 168 <-> COM RxPDO-Map Outputs Channel 2/Data Out 21
//     SerialComm Outputs/GVL_SDS.PCMB.stSerial2.stComOut/D @bit 24 <-> COM RxPDO-Map Outputs Channel 2/Data Out 3
//     SerialComm Outputs/GVL_SDS.PCMB.stSerial2.stComOut/D @bit 32 <-> COM RxPDO-Map Outputs Channel 2/Data Out 4
//     SerialComm Outputs/GVL_SDS.PCMB.stSerial2.stComOut/D @bit 40 <-> COM RxPDO-Map Outputs Channel 2/Data Out 5
//     SerialComm Outputs/GVL_SDS.PCMB.stSerial2.stComOut/D @bit 48 <-> COM RxPDO-Map Outputs Channel 2/Data Out 6
//     SerialComm Outputs/GVL_SDS.PCMB.stSerial2.stComOut/D @bit 56 <-> COM RxPDO-Map Outputs Channel 2/Data Out 7
//     SerialComm Outputs/GVL_SDS.PCMB.stSerial2.stComOut/D @bit 64 <-> COM RxPDO-Map Outputs Channel 2/Data Out 8
//     SerialComm Outputs/GVL_SDS.PCMB.stSerial2.stComOut/D @bit 72 <-> COM RxPDO-Map Outputs Channel 2/Data Out 9
//   sample_delivery Instance <-> MAIN (EtherCAT)/PCM C (EP1111)
//     PlcTask Inputs/GVL_SDS.PCMC.stBaseIO.i_SyncUnitWC <-> WcState/WcState
//   sample_delivery Instance <-> MAIN (EtherCAT)/PCM C (EP4374-0002)
//     PlcTask Inputs/GVL_SDS.PCMC.stPropAir1.i_iPressRB <-> AI Inputs Channel 1/Value
//     PlcTask Inputs/GVL_SDS.PCMC.stPropAir2.i_iPressRB <-> AI Inputs Channel 2/Value
//     PlcTask Outputs/GVL_SDS.PCMC.stPropAir1.q_iPressCt <-> AO Outputs Channel 3/Analog output
//     PlcTask Outputs/GVL_SDS.PCMC.stPropAir2.q_iPressCt <-> AO Outputs Channel 4/Analog output
//   sample_delivery Instance <-> MAIN (EtherCAT)/PCM C (EP6002-0002)
//     SerialComm Inputs/GVL_SDS.PCMC.stSerial1.stComIn/D <-> COM TxPDO-Map Inputs Channel 1/Data In 0
//     SerialComm Inputs/GVL_SDS.PCMC.stSerial2.stComIn/D <-> COM TxPDO-Map Inputs Channel 2/Data In 0
//     SerialComm Inputs/GVL_SDS.PCMC.stSerial1.stComIn/D @bit 8 <-> COM TxPDO-Map Inputs Channel 1/Data In 1
//     SerialComm Inputs/GVL_SDS.PCMC.stSerial1.stComIn/D @bit 80 <-> COM TxPDO-Map Inputs Channel 1/Data In 10
//     SerialComm Inputs/GVL_SDS.PCMC.stSerial1.stComIn/D @bit 88 <-> COM TxPDO-Map Inputs Channel 1/Data In 11
//     SerialComm Inputs/GVL_SDS.PCMC.stSerial1.stComIn/D @bit 96 <-> COM TxPDO-Map Inputs Channel 1/Data In 12
//     SerialComm Inputs/GVL_SDS.PCMC.stSerial1.stComIn/D @bit 104 <-> COM TxPDO-Map Inputs Channel 1/Data In 13
//     SerialComm Inputs/GVL_SDS.PCMC.stSerial1.stComIn/D @bit 112 <-> COM TxPDO-Map Inputs Channel 1/Data In 14
//     SerialComm Inputs/GVL_SDS.PCMC.stSerial1.stComIn/D @bit 120 <-> COM TxPDO-Map Inputs Channel 1/Data In 15
//     SerialComm Inputs/GVL_SDS.PCMC.stSerial1.stComIn/D @bit 128 <-> COM TxPDO-Map Inputs Channel 1/Data In 16
//     SerialComm Inputs/GVL_SDS.PCMC.stSerial1.stComIn/D @bit 136 <-> COM TxPDO-Map Inputs Channel 1/Data In 17
//     SerialComm Inputs/GVL_SDS.PCMC.stSerial1.stComIn/D @bit 144 <-> COM TxPDO-Map Inputs Channel 1/Data In 18
//     SerialComm Inputs/GVL_SDS.PCMC.stSerial1.stComIn/D @bit 152 <-> COM TxPDO-Map Inputs Channel 1/Data In 19
//     SerialComm Inputs/GVL_SDS.PCMC.stSerial1.stComIn/D @bit 16 <-> COM TxPDO-Map Inputs Channel 1/Data In 2
//     SerialComm Inputs/GVL_SDS.PCMC.stSerial1.stComIn/D @bit 160 <-> COM TxPDO-Map Inputs Channel 1/Data In 20
//     SerialComm Inputs/GVL_SDS.PCMC.stSerial1.stComIn/D @bit 168 <-> COM TxPDO-Map Inputs Channel 1/Data In 21
//     SerialComm Inputs/GVL_SDS.PCMC.stSerial1.stComIn/D @bit 24 <-> COM TxPDO-Map Inputs Channel 1/Data In 3
//     SerialComm Inputs/GVL_SDS.PCMC.stSerial1.stComIn/D @bit 32 <-> COM TxPDO-Map Inputs Channel 1/Data In 4
//     SerialComm Inputs/GVL_SDS.PCMC.stSerial1.stComIn/D @bit 40 <-> COM TxPDO-Map Inputs Channel 1/Data In 5
//     SerialComm Inputs/GVL_SDS.PCMC.stSerial1.stComIn/D @bit 48 <-> COM TxPDO-Map Inputs Channel 1/Data In 6
//     SerialComm Inputs/GVL_SDS.PCMC.stSerial1.stComIn/D @bit 56 <-> COM TxPDO-Map Inputs Channel 1/Data In 7
//     SerialComm Inputs/GVL_SDS.PCMC.stSerial1.stComIn/D @bit 64 <-> COM TxPDO-Map Inputs Channel 1/Data In 8
//     SerialComm Inputs/GVL_SDS.PCMC.stSerial1.stComIn/D @bit 72 <-> COM TxPDO-Map Inputs Channel 1/Data In 9
//     SerialComm Inputs/GVL_SDS.PCMC.stSerial2.stComIn/D @bit 8 <-> COM TxPDO-Map Inputs Channel 2/Data In 1
//     SerialComm Inputs/GVL_SDS.PCMC.stSerial2.stComIn/D @bit 80 <-> COM TxPDO-Map Inputs Channel 2/Data In 10
//     SerialComm Inputs/GVL_SDS.PCMC.stSerial2.stComIn/D @bit 88 <-> COM TxPDO-Map Inputs Channel 2/Data In 11
//     SerialComm Inputs/GVL_SDS.PCMC.stSerial2.stComIn/D @bit 96 <-> COM TxPDO-Map Inputs Channel 2/Data In 12
//     SerialComm Inputs/GVL_SDS.PCMC.stSerial2.stComIn/D @bit 104 <-> COM TxPDO-Map Inputs Channel 2/Data In 13
//     SerialComm Inputs/GVL_SDS.PCMC.stSerial2.stComIn/D @bit 112 <-> COM TxPDO-Map Inputs Channel 2/Data In 14
//     SerialComm Inputs/GVL_SDS.PCMC.stSerial2.stComIn/D @bit 120 <-> COM TxPDO-Map Inputs Channel 2/Data In 15
//     SerialComm Inputs/GVL_SDS.PCMC.stSerial2.stComIn/D @bit 128 <-> COM TxPDO-Map Inputs Channel 2/Data In 16
//     SerialComm Inputs/GVL_SDS.PCMC.stSerial2.stComIn/D @bit 136 <-> COM TxPDO-Map Inputs Channel 2/Data In 17
//     SerialComm Inputs/GVL_SDS.PCMC.stSerial2.stComIn/D @bit 144 <-> COM TxPDO-Map Inputs Channel 2/Data In 18
//     SerialComm Inputs/GVL_SDS.PCMC.stSerial2.stComIn/D @bit 152 <-> COM TxPDO-Map Inputs Channel 2/Data In 19
//     SerialComm Inputs/GVL_SDS.PCMC.stSerial2.stComIn/D @bit 16 <-> COM TxPDO-Map Inputs Channel 2/Data In 2
//     SerialComm Inputs/GVL_SDS.PCMC.stSerial2.stComIn/D @bit 160 <-> COM TxPDO-Map Inputs Channel 2/Data In 20
//     SerialComm Inputs/GVL_SDS.PCMC.stSerial2.stComIn/D @bit 168 <-> COM TxPDO-Map Inputs Channel 2/Data In 21
//     SerialComm Inputs/GVL_SDS.PCMC.stSerial2.stComIn/D @bit 24 <-> COM TxPDO-Map Inputs Channel 2/Data In 3
//     SerialComm Inputs/GVL_SDS.PCMC.stSerial2.stComIn/D @bit 32 <-> COM TxPDO-Map Inputs Channel 2/Data In 4
//     SerialComm Inputs/GVL_SDS.PCMC.stSerial2.stComIn/D @bit 40 <-> COM TxPDO-Map Inputs Channel 2/Data In 5
//     SerialComm Inputs/GVL_SDS.PCMC.stSerial2.stComIn/D @bit 48 <-> COM TxPDO-Map Inputs Channel 2/Data In 6
//     SerialComm Inputs/GVL_SDS.PCMC.stSerial2.stComIn/D @bit 56 <-> COM TxPDO-Map Inputs Channel 2/Data In 7
//     SerialComm Inputs/GVL_SDS.PCMC.stSerial2.stComIn/D @bit 64 <-> COM TxPDO-Map Inputs Channel 2/Data In 8
//     SerialComm Inputs/GVL_SDS.PCMC.stSerial2.stComIn/D @bit 72 <-> COM TxPDO-Map Inputs Channel 2/Data In 9
//     SerialComm Inputs/GVL_SDS.PCMC.stSerial1.stComIn/Status <-> COM TxPDO-Map Inputs Channel 1/Status
//     SerialComm Inputs/GVL_SDS.PCMC.stSerial2.stComIn/Status <-> COM TxPDO-Map Inputs Channel 2/Status
//     SerialComm Outputs/GVL_SDS.PCMC.stSerial1.stComOut/Ctrl <-> COM RxPDO-Map Outputs Channel 1/Ctrl
//     SerialComm Outputs/GVL_SDS.PCMC.stSerial2.stComOut/Ctrl <-> COM RxPDO-Map Outputs Channel 2/Ctrl
//     SerialComm Outputs/GVL_SDS.PCMC.stSerial1.stComOut/D <-> COM RxPDO-Map Outputs Channel 1/Data Out 0
//     SerialComm Outputs/GVL_SDS.PCMC.stSerial2.stComOut/D <-> COM RxPDO-Map Outputs Channel 2/Data Out 0
//     SerialComm Outputs/GVL_SDS.PCMC.stSerial1.stComOut/D @bit 8 <-> COM RxPDO-Map Outputs Channel 1/Data Out 1
//     SerialComm Outputs/GVL_SDS.PCMC.stSerial1.stComOut/D @bit 80 <-> COM RxPDO-Map Outputs Channel 1/Data Out 10
//     SerialComm Outputs/GVL_SDS.PCMC.stSerial1.stComOut/D @bit 88 <-> COM RxPDO-Map Outputs Channel 1/Data Out 11
//     SerialComm Outputs/GVL_SDS.PCMC.stSerial1.stComOut/D @bit 96 <-> COM RxPDO-Map Outputs Channel 1/Data Out 12
//     SerialComm Outputs/GVL_SDS.PCMC.stSerial1.stComOut/D @bit 104 <-> COM RxPDO-Map Outputs Channel 1/Data Out 13
//     SerialComm Outputs/GVL_SDS.PCMC.stSerial1.stComOut/D @bit 112 <-> COM RxPDO-Map Outputs Channel 1/Data Out 14
//     SerialComm Outputs/GVL_SDS.PCMC.stSerial1.stComOut/D @bit 120 <-> COM RxPDO-Map Outputs Channel 1/Data Out 15
//     SerialComm Outputs/GVL_SDS.PCMC.stSerial1.stComOut/D @bit 128 <-> COM RxPDO-Map Outputs Channel 1/Data Out 16
//     SerialComm Outputs/GVL_SDS.PCMC.stSerial1.stComOut/D @bit 136 <-> COM RxPDO-Map Outputs Channel 1/Data Out 17
//     SerialComm Outputs/GVL_SDS.PCMC.stSerial1.stComOut/D @bit 144 <-> COM RxPDO-Map Outputs Channel 1/Data Out 18
//     SerialComm Outputs/GVL_SDS.PCMC.stSerial1.stComOut/D @bit 152 <-> COM RxPDO-Map Outputs Channel 1/Data Out 19
//     SerialComm Outputs/GVL_SDS.PCMC.stSerial1.stComOut/D @bit 16 <-> COM RxPDO-Map Outputs Channel 1/Data Out 2
//     SerialComm Outputs/GVL_SDS.PCMC.stSerial1.stComOut/D @bit 160 <-> COM RxPDO-Map Outputs Channel 1/Data Out 20
//     SerialComm Outputs/GVL_SDS.PCMC.stSerial1.stComOut/D @bit 168 <-> COM RxPDO-Map Outputs Channel 1/Data Out 21
//     SerialComm Outputs/GVL_SDS.PCMC.stSerial1.stComOut/D @bit 24 <-> COM RxPDO-Map Outputs Channel 1/Data Out 3
//     SerialComm Outputs/GVL_SDS.PCMC.stSerial1.stComOut/D @bit 32 <-> COM RxPDO-Map Outputs Channel 1/Data Out 4
//     SerialComm Outputs/GVL_SDS.PCMC.stSerial1.stComOut/D @bit 40 <-> COM RxPDO-Map Outputs Channel 1/Data Out 5
//     SerialComm Outputs/GVL_SDS.PCMC.stSerial1.stComOut/D @bit 48 <-> COM RxPDO-Map Outputs Channel 1/Data Out 6
//     SerialComm Outputs/GVL_SDS.PCMC.stSerial1.stComOut/D @bit 56 <-> COM RxPDO-Map Outputs Channel 1/Data Out 7
//     SerialComm Outputs/GVL_SDS.PCMC.stSerial1.stComOut/D @bit 64 <-> COM RxPDO-Map Outputs Channel 1/Data Out 8
//     SerialComm Outputs/GVL_SDS.PCMC.stSerial1.stComOut/D @bit 72 <-> COM RxPDO-Map Outputs Channel 1/Data Out 9
//     SerialComm Outputs/GVL_SDS.PCMC.stSerial2.stComOut/D @bit 8 <-> COM RxPDO-Map Outputs Channel 2/Data Out 1
//     SerialComm Outputs/GVL_SDS.PCMC.stSerial2.stComOut/D @bit 80 <-> COM RxPDO-Map Outputs Channel 2/Data Out 10
//     SerialComm Outputs/GVL_SDS.PCMC.stSerial2.stComOut/D @bit 88 <-> COM RxPDO-Map Outputs Channel 2/Data Out 11
//     SerialComm Outputs/GVL_SDS.PCMC.stSerial2.stComOut/D @bit 96 <-> COM RxPDO-Map Outputs Channel 2/Data Out 12
//     SerialComm Outputs/GVL_SDS.PCMC.stSerial2.stComOut/D @bit 104 <-> COM RxPDO-Map Outputs Channel 2/Data Out 13
//     SerialComm Outputs/GVL_SDS.PCMC.stSerial2.stComOut/D @bit 112 <-> COM RxPDO-Map Outputs Channel 2/Data Out 14
//     SerialComm Outputs/GVL_SDS.PCMC.stSerial2.stComOut/D @bit 120 <-> COM RxPDO-Map Outputs Channel 2/Data Out 15
//     SerialComm Outputs/GVL_SDS.PCMC.stSerial2.stComOut/D @bit 128 <-> COM RxPDO-Map Outputs Channel 2/Data Out 16
//     SerialComm Outputs/GVL_SDS.PCMC.stSerial2.stComOut/D @bit 136 <-> COM RxPDO-Map Outputs Channel 2/Data Out 17
//     SerialComm Outputs/GVL_SDS.PCMC.stSerial2.stComOut/D @bit 144 <-> COM RxPDO-Map Outputs Channel 2/Data Out 18
//     SerialComm Outputs/GVL_SDS.PCMC.stSerial2.stComOut/D @bit 152 <-> COM RxPDO-Map Outputs Channel 2/Data Out 19
//     SerialComm Outputs/GVL_SDS.PCMC.stSerial2.stComOut/D @bit 16 <-> COM RxPDO-Map Outputs Channel 2/Data Out 2
//     SerialComm Outputs/GVL_SDS.PCMC.stSerial2.stComOut/D @bit 160 <-> COM RxPDO-Map Outputs Channel 2/Data Out 20
//     SerialComm Outputs/GVL_SDS.PCMC.stSerial2.stComOut/D @bit 168 <-> COM RxPDO-Map Outputs Channel 2/Data Out 21
//     SerialComm Outputs/GVL_SDS.PCMC.stSerial2.stComOut/D @bit 24 <-> COM RxPDO-Map Outputs Channel 2/Data Out 3
//     SerialComm Outputs/GVL_SDS.PCMC.stSerial2.stComOut/D @bit 32 <-> COM RxPDO-Map Outputs Channel 2/Data Out 4
//     SerialComm Outputs/GVL_SDS.PCMC.stSerial2.stComOut/D @bit 40 <-> COM RxPDO-Map Outputs Channel 2/Data Out 5
//     SerialComm Outputs/GVL_SDS.PCMC.stSerial2.stComOut/D @bit 48 <-> COM RxPDO-Map Outputs Channel 2/Data Out 6
//     SerialComm Outputs/GVL_SDS.PCMC.stSerial2.stComOut/D @bit 56 <-> COM RxPDO-Map Outputs Channel 2/Data Out 7
//     SerialComm Outputs/GVL_SDS.PCMC.stSerial2.stComOut/D @bit 64 <-> COM RxPDO-Map Outputs Channel 2/Data Out 8
//     SerialComm Outputs/GVL_SDS.PCMC.stSerial2.stComOut/D @bit 72 <-> COM RxPDO-Map Outputs Channel 2/Data Out 9
//   sample_delivery Instance <-> MAIN (EtherCAT)/PCM D (EP1111)
//     PlcTask Inputs/GVL_SDS.PCMD.stBaseIO.i_SyncUnitWC <-> WcState/WcState
//   sample_delivery Instance <-> MAIN (EtherCAT)/PCM D (EP4374-0002)
//     PlcTask Inputs/GVL_SDS.PCMD.stPropAir1.i_iPressRB <-> AI Inputs Channel 1/Value
//     PlcTask Inputs/GVL_SDS.PCMD.stPropAir2.i_iPressRB <-> AI Inputs Channel 2/Value
//     PlcTask Outputs/GVL_SDS.PCMD.stPropAir1.q_iPressCt <-> AO Outputs Channel 3/Analog output
//     PlcTask Outputs/GVL_SDS.PCMD.stPropAir2.q_iPressCt <-> AO Outputs Channel 4/Analog output
//   sample_delivery Instance <-> MAIN (EtherCAT)/PCM D (EP6002-0002)
//     SerialComm Inputs/GVL_SDS.PCMD.stSerial1.stComIn/D <-> COM TxPDO-Map Inputs Channel 1/Data In 0
//     SerialComm Inputs/GVL_SDS.PCMD.stSerial2.stComIn/D <-> COM TxPDO-Map Inputs Channel 2/Data In 0
//     SerialComm Inputs/GVL_SDS.PCMD.stSerial1.stComIn/D @bit 8 <-> COM TxPDO-Map Inputs Channel 1/Data In 1
//     SerialComm Inputs/GVL_SDS.PCMD.stSerial1.stComIn/D @bit 80 <-> COM TxPDO-Map Inputs Channel 1/Data In 10
//     SerialComm Inputs/GVL_SDS.PCMD.stSerial1.stComIn/D @bit 88 <-> COM TxPDO-Map Inputs Channel 1/Data In 11
//     SerialComm Inputs/GVL_SDS.PCMD.stSerial1.stComIn/D @bit 96 <-> COM TxPDO-Map Inputs Channel 1/Data In 12
//     SerialComm Inputs/GVL_SDS.PCMD.stSerial1.stComIn/D @bit 104 <-> COM TxPDO-Map Inputs Channel 1/Data In 13
//     SerialComm Inputs/GVL_SDS.PCMD.stSerial1.stComIn/D @bit 112 <-> COM TxPDO-Map Inputs Channel 1/Data In 14
//     SerialComm Inputs/GVL_SDS.PCMD.stSerial1.stComIn/D @bit 120 <-> COM TxPDO-Map Inputs Channel 1/Data In 15
//     SerialComm Inputs/GVL_SDS.PCMD.stSerial1.stComIn/D @bit 128 <-> COM TxPDO-Map Inputs Channel 1/Data In 16
//     SerialComm Inputs/GVL_SDS.PCMD.stSerial1.stComIn/D @bit 136 <-> COM TxPDO-Map Inputs Channel 1/Data In 17
//     SerialComm Inputs/GVL_SDS.PCMD.stSerial1.stComIn/D @bit 144 <-> COM TxPDO-Map Inputs Channel 1/Data In 18
//     SerialComm Inputs/GVL_SDS.PCMD.stSerial1.stComIn/D @bit 152 <-> COM TxPDO-Map Inputs Channel 1/Data In 19
//     SerialComm Inputs/GVL_SDS.PCMD.stSerial1.stComIn/D @bit 16 <-> COM TxPDO-Map Inputs Channel 1/Data In 2
//     SerialComm Inputs/GVL_SDS.PCMD.stSerial1.stComIn/D @bit 160 <-> COM TxPDO-Map Inputs Channel 1/Data In 20
//     SerialComm Inputs/GVL_SDS.PCMD.stSerial1.stComIn/D @bit 168 <-> COM TxPDO-Map Inputs Channel 1/Data In 21
//     SerialComm Inputs/GVL_SDS.PCMD.stSerial1.stComIn/D @bit 24 <-> COM TxPDO-Map Inputs Channel 1/Data In 3
//     SerialComm Inputs/GVL_SDS.PCMD.stSerial1.stComIn/D @bit 32 <-> COM TxPDO-Map Inputs Channel 1/Data In 4
//     SerialComm Inputs/GVL_SDS.PCMD.stSerial1.stComIn/D @bit 40 <-> COM TxPDO-Map Inputs Channel 1/Data In 5
//     SerialComm Inputs/GVL_SDS.PCMD.stSerial1.stComIn/D @bit 48 <-> COM TxPDO-Map Inputs Channel 1/Data In 6
//     SerialComm Inputs/GVL_SDS.PCMD.stSerial1.stComIn/D @bit 56 <-> COM TxPDO-Map Inputs Channel 1/Data In 7
//     SerialComm Inputs/GVL_SDS.PCMD.stSerial1.stComIn/D @bit 64 <-> COM TxPDO-Map Inputs Channel 1/Data In 8
//     SerialComm Inputs/GVL_SDS.PCMD.stSerial1.stComIn/D @bit 72 <-> COM TxPDO-Map Inputs Channel 1/Data In 9
//     SerialComm Inputs/GVL_SDS.PCMD.stSerial2.stComIn/D @bit 8 <-> COM TxPDO-Map Inputs Channel 2/Data In 1
//     SerialComm Inputs/GVL_SDS.PCMD.stSerial2.stComIn/D @bit 80 <-> COM TxPDO-Map Inputs Channel 2/Data In 10
//     SerialComm Inputs/GVL_SDS.PCMD.stSerial2.stComIn/D @bit 88 <-> COM TxPDO-Map Inputs Channel 2/Data In 11
//     SerialComm Inputs/GVL_SDS.PCMD.stSerial2.stComIn/D @bit 96 <-> COM TxPDO-Map Inputs Channel 2/Data In 12
//     SerialComm Inputs/GVL_SDS.PCMD.stSerial2.stComIn/D @bit 104 <-> COM TxPDO-Map Inputs Channel 2/Data In 13
//     SerialComm Inputs/GVL_SDS.PCMD.stSerial2.stComIn/D @bit 112 <-> COM TxPDO-Map Inputs Channel 2/Data In 14
//     SerialComm Inputs/GVL_SDS.PCMD.stSerial2.stComIn/D @bit 120 <-> COM TxPDO-Map Inputs Channel 2/Data In 15
//     SerialComm Inputs/GVL_SDS.PCMD.stSerial2.stComIn/D @bit 128 <-> COM TxPDO-Map Inputs Channel 2/Data In 16
//     SerialComm Inputs/GVL_SDS.PCMD.stSerial2.stComIn/D @bit 136 <-> COM TxPDO-Map Inputs Channel 2/Data In 17
//     SerialComm Inputs/GVL_SDS.PCMD.stSerial2.stComIn/D @bit 144 <-> COM TxPDO-Map Inputs Channel 2/Data In 18
//     SerialComm Inputs/GVL_SDS.PCMD.stSerial2.stComIn/D @bit 152 <-> COM TxPDO-Map Inputs Channel 2/Data In 19
//     SerialComm Inputs/GVL_SDS.PCMD.stSerial2.stComIn/D @bit 16 <-> COM TxPDO-Map Inputs Channel 2/Data In 2
//     SerialComm Inputs/GVL_SDS.PCMD.stSerial2.stComIn/D @bit 160 <-> COM TxPDO-Map Inputs Channel 2/Data In 20
//     SerialComm Inputs/GVL_SDS.PCMD.stSerial2.stComIn/D @bit 168 <-> COM TxPDO-Map Inputs Channel 2/Data In 21
//     SerialComm Inputs/GVL_SDS.PCMD.stSerial2.stComIn/D @bit 24 <-> COM TxPDO-Map Inputs Channel 2/Data In 3
//     SerialComm Inputs/GVL_SDS.PCMD.stSerial2.stComIn/D @bit 32 <-> COM TxPDO-Map Inputs Channel 2/Data In 4
//     SerialComm Inputs/GVL_SDS.PCMD.stSerial2.stComIn/D @bit 40 <-> COM TxPDO-Map Inputs Channel 2/Data In 5
//     SerialComm Inputs/GVL_SDS.PCMD.stSerial2.stComIn/D @bit 48 <-> COM TxPDO-Map Inputs Channel 2/Data In 6
//     SerialComm Inputs/GVL_SDS.PCMD.stSerial2.stComIn/D @bit 56 <-> COM TxPDO-Map Inputs Channel 2/Data In 7
//     SerialComm Inputs/GVL_SDS.PCMD.stSerial2.stComIn/D @bit 64 <-> COM TxPDO-Map Inputs Channel 2/Data In 8
//     SerialComm Inputs/GVL_SDS.PCMD.stSerial2.stComIn/D @bit 72 <-> COM TxPDO-Map Inputs Channel 2/Data In 9
//     SerialComm Inputs/GVL_SDS.PCMD.stSerial1.stComIn/Status <-> COM TxPDO-Map Inputs Channel 1/Status
//     SerialComm Inputs/GVL_SDS.PCMD.stSerial2.stComIn/Status <-> COM TxPDO-Map Inputs Channel 2/Status
//     SerialComm Outputs/GVL_SDS.PCMD.stSerial1.stComOut/Ctrl <-> COM RxPDO-Map Outputs Channel 1/Ctrl
//     SerialComm Outputs/GVL_SDS.PCMD.stSerial2.stComOut/Ctrl <-> COM RxPDO-Map Outputs Channel 2/Ctrl
//     SerialComm Outputs/GVL_SDS.PCMD.stSerial1.stComOut/D <-> COM RxPDO-Map Outputs Channel 1/Data Out 0
//     SerialComm Outputs/GVL_SDS.PCMD.stSerial2.stComOut/D <-> COM RxPDO-Map Outputs Channel 2/Data Out 0
//     SerialComm Outputs/GVL_SDS.PCMD.stSerial1.stComOut/D @bit 8 <-> COM RxPDO-Map Outputs Channel 1/Data Out 1
//     SerialComm Outputs/GVL_SDS.PCMD.stSerial1.stComOut/D @bit 80 <-> COM RxPDO-Map Outputs Channel 1/Data Out 10
//     SerialComm Outputs/GVL_SDS.PCMD.stSerial1.stComOut/D @bit 88 <-> COM RxPDO-Map Outputs Channel 1/Data Out 11
//     SerialComm Outputs/GVL_SDS.PCMD.stSerial1.stComOut/D @bit 96 <-> COM RxPDO-Map Outputs Channel 1/Data Out 12
//     SerialComm Outputs/GVL_SDS.PCMD.stSerial1.stComOut/D @bit 104 <-> COM RxPDO-Map Outputs Channel 1/Data Out 13
//     SerialComm Outputs/GVL_SDS.PCMD.stSerial1.stComOut/D @bit 112 <-> COM RxPDO-Map Outputs Channel 1/Data Out 14
//     SerialComm Outputs/GVL_SDS.PCMD.stSerial1.stComOut/D @bit 120 <-> COM RxPDO-Map Outputs Channel 1/Data Out 15
//     SerialComm Outputs/GVL_SDS.PCMD.stSerial1.stComOut/D @bit 128 <-> COM RxPDO-Map Outputs Channel 1/Data Out 16
//     SerialComm Outputs/GVL_SDS.PCMD.stSerial1.stComOut/D @bit 136 <-> COM RxPDO-Map Outputs Channel 1/Data Out 17
//     SerialComm Outputs/GVL_SDS.PCMD.stSerial1.stComOut/D @bit 144 <-> COM RxPDO-Map Outputs Channel 1/Data Out 18
//     SerialComm Outputs/GVL_SDS.PCMD.stSerial1.stComOut/D @bit 152 <-> COM RxPDO-Map Outputs Channel 1/Data Out 19
//     SerialComm Outputs/GVL_SDS.PCMD.stSerial1.stComOut/D @bit 16 <-> COM RxPDO-Map Outputs Channel 1/Data Out 2
//     SerialComm Outputs/GVL_SDS.PCMD.stSerial1.stComOut/D @bit 160 <-> COM RxPDO-Map Outputs Channel 1/Data Out 20
//     SerialComm Outputs/GVL_SDS.PCMD.stSerial1.stComOut/D @bit 168 <-> COM RxPDO-Map Outputs Channel 1/Data Out 21
//     SerialComm Outputs/GVL_SDS.PCMD.stSerial1.stComOut/D @bit 24 <-> COM RxPDO-Map Outputs Channel 1/Data Out 3
//     SerialComm Outputs/GVL_SDS.PCMD.stSerial1.stComOut/D @bit 32 <-> COM RxPDO-Map Outputs Channel 1/Data Out 4
//     SerialComm Outputs/GVL_SDS.PCMD.stSerial1.stComOut/D @bit 40 <-> COM RxPDO-Map Outputs Channel 1/Data Out 5
//     SerialComm Outputs/GVL_SDS.PCMD.stSerial1.stComOut/D @bit 48 <-> COM RxPDO-Map Outputs Channel 1/Data Out 6
//     SerialComm Outputs/GVL_SDS.PCMD.stSerial1.stComOut/D @bit 56 <-> COM RxPDO-Map Outputs Channel 1/Data Out 7
//     SerialComm Outputs/GVL_SDS.PCMD.stSerial1.stComOut/D @bit 64 <-> COM RxPDO-Map Outputs Channel 1/Data Out 8
//     SerialComm Outputs/GVL_SDS.PCMD.stSerial1.stComOut/D @bit 72 <-> COM RxPDO-Map Outputs Channel 1/Data Out 9
//     SerialComm Outputs/GVL_SDS.PCMD.stSerial2.stComOut/D @bit 8 <-> COM RxPDO-Map Outputs Channel 2/Data Out 1
//     SerialComm Outputs/GVL_SDS.PCMD.stSerial2.stComOut/D @bit 80 <-> COM RxPDO-Map Outputs Channel 2/Data Out 10
//     SerialComm Outputs/GVL_SDS.PCMD.stSerial2.stComOut/D @bit 88 <-> COM RxPDO-Map Outputs Channel 2/Data Out 11
//     SerialComm Outputs/GVL_SDS.PCMD.stSerial2.stComOut/D @bit 96 <-> COM RxPDO-Map Outputs Channel 2/Data Out 12
//     SerialComm Outputs/GVL_SDS.PCMD.stSerial2.stComOut/D @bit 104 <-> COM RxPDO-Map Outputs Channel 2/Data Out 13
//     SerialComm Outputs/GVL_SDS.PCMD.stSerial2.stComOut/D @bit 112 <-> COM RxPDO-Map Outputs Channel 2/Data Out 14
//     SerialComm Outputs/GVL_SDS.PCMD.stSerial2.stComOut/D @bit 120 <-> COM RxPDO-Map Outputs Channel 2/Data Out 15
//     SerialComm Outputs/GVL_SDS.PCMD.stSerial2.stComOut/D @bit 128 <-> COM RxPDO-Map Outputs Channel 2/Data Out 16
//     SerialComm Outputs/GVL_SDS.PCMD.stSerial2.stComOut/D @bit 136 <-> COM RxPDO-Map Outputs Channel 2/Data Out 17
//     SerialComm Outputs/GVL_SDS.PCMD.stSerial2.stComOut/D @bit 144 <-> COM RxPDO-Map Outputs Channel 2/Data Out 18
//     SerialComm Outputs/GVL_SDS.PCMD.stSerial2.stComOut/D @bit 152 <-> COM RxPDO-Map Outputs Channel 2/Data Out 19
//     SerialComm Outputs/GVL_SDS.PCMD.stSerial2.stComOut/D @bit 16 <-> COM RxPDO-Map Outputs Channel 2/Data Out 2
//     SerialComm Outputs/GVL_SDS.PCMD.stSerial2.stComOut/D @bit 160 <-> COM RxPDO-Map Outputs Channel 2/Data Out 20
//     SerialComm Outputs/GVL_SDS.PCMD.stSerial2.stComOut/D @bit 168 <-> COM RxPDO-Map Outputs Channel 2/Data Out 21
//     SerialComm Outputs/GVL_SDS.PCMD.stSerial2.stComOut/D @bit 24 <-> COM RxPDO-Map Outputs Channel 2/Data Out 3
//     SerialComm Outputs/GVL_SDS.PCMD.stSerial2.stComOut/D @bit 32 <-> COM RxPDO-Map Outputs Channel 2/Data Out 4
//     SerialComm Outputs/GVL_SDS.PCMD.stSerial2.stComOut/D @bit 40 <-> COM RxPDO-Map Outputs Channel 2/Data Out 5
//     SerialComm Outputs/GVL_SDS.PCMD.stSerial2.stComOut/D @bit 48 <-> COM RxPDO-Map Outputs Channel 2/Data Out 6
//     SerialComm Outputs/GVL_SDS.PCMD.stSerial2.stComOut/D @bit 56 <-> COM RxPDO-Map Outputs Channel 2/Data Out 7
//     SerialComm Outputs/GVL_SDS.PCMD.stSerial2.stComOut/D @bit 64 <-> COM RxPDO-Map Outputs Channel 2/Data Out 8
//     SerialComm Outputs/GVL_SDS.PCMD.stSerial2.stComOut/D @bit 72 <-> COM RxPDO-Map Outputs Channel 2/Data Out 9
//   sample_delivery Instance <-> MAIN (EtherCAT)/Solenoid Pair A Digital IO (EP2338-0001)
//     PlcTask Outputs/GVL_SDS.SolenoidPairA.q_xDO1 <-> Channel 9/Output
//     PlcTask Outputs/GVL_SDS.SolenoidPairA.q_xDO2 <-> Channel 10/Output

// ---- GVLs/GVL_SDS.TcGVL
VAR_GLOBAL
{attribute 'pytmc' := 'pv: ICL:SDS:SEL:A'}
{attribute 'TcLinkTo' := '.stSensSerial.stComIn.Status := TIIB[M3 Selector A Serial IO (EP6002-0002)]^COM TxPDO-Map Inputs Channel 1^Status;
                          .stViciSerial.stComIn.Status := TIIB[M3 Selector A Serial IO (EP6002-0002)]^COM TxPDO-Map Inputs Channel 2^Status;
                          .stSensSerial.stComOut.Ctrl := TIID^MAIN (EtherCAT)^M3 Selector A Serial IO (EP6002-0002)^COM RxPDO-Map Outputs Channel 1^Ctrl;
                          .stViciSerial.stComOut.Ctrl := TIID^MAIN (EtherCAT)^M3 Selector A Serial IO (EP6002-0002)^COM RxPDO-Map Outputs Channel 2^Ctrl;
                          .stShaker01.q_xPwrDO := TIIB[M3 Selector A Digital IO (EP2338-1001)]^Channel 9^Output;
                          .stShaker02.q_xPwrDO := TIIB[M3 Selector A Digital IO (EP2338-1001)]^Channel 10^Output;
                          .stShaker03.q_xPwrDO := TIIB[M3 Selector A Digital IO (EP2338-1001)]^Channel 11^Output;
                          .stShaker04.q_xPwrDO := TIIB[M3 Selector A Digital IO (EP2338-1001)]^Channel 12^Output;
                          .stBaseIO.i_SyncUnitWC := TIID^MAIN (EtherCAT)^M3 Selector A (EP1111)^WcState^WcState;
'}
M3SelectorA : FB_SelectorM3;

{attribute 'pytmc' := 'pv: ICL:SDS:SEL:B'}
{attribute 'TcLinkTo' := '.stSensSerial.stComIn.Status := TIIB[M3 Selector B Serial IO (EP6002-0002)]^COM TxPDO-Map Inputs Channel 1^Status;
                          .stViciSerial.stComIn.Status := TIIB[M3 Selector B Serial IO (EP6002-0002)]^COM TxPDO-Map Inputs Channel 2^Status;
                          .stSensSerial.stComOut.Ctrl := TIID^MAIN (EtherCAT)^M3 Selector B Serial IO (EP6002-0002)^COM RxPDO-Map Outputs Channel 1^Ctrl;
                          .stViciSerial.stComOut.Ctrl := TIID^MAIN (EtherCAT)^M3 Selector B Serial IO (EP6002-0002)^COM RxPDO-Map Outputs Channel 2^Ctrl;
                          .stShaker01.q_xPwrDO := TIIB[M3 Selector B Digital IO (EP2338-1001)]^Channel 9^Output;
                          .stShaker02.q_xPwrDO := TIIB[M3 Selector B Digital IO (EP2338-1001)]^Channel 10^Output;
                          .stShaker03.q_xPwrDO := TIIB[M3 Selector B Digital IO (EP2338-1001)]^Channel 11^Output;
                          .stShaker04.q_xPwrDO := TIIB[M3 Selector B Digital IO (EP2338-1001)]^Channel 12^Output;
                          .stBaseIO.i_SyncUnitWC := TIID^MAIN (EtherCAT)^M3 Selector B (EP1111)^WcState^WcState
'}
M3SelectorB : FB_SelectorM3;

{attribute 'pytmc' := 'pv: ICL:SDS:SEL:C'}
{attribute 'TcLinkTo' := '.stSensSerial.stComIn.Status := TIIB[M3 Selector C Serial IO (EP6002-0002)]^COM TxPDO-Map Inputs Channel 1^Status;
                          .stViciSerial.stComIn.Status := TIIB[M3 Selector C Serial IO (EP6002-0002)]^COM TxPDO-Map Inputs Channel 2^Status;
                          .stSensSerial.stComOut.Ctrl := TIID^MAIN (EtherCAT)^M3 Selector C Serial IO (EP6002-0002)^COM RxPDO-Map Outputs Channel 1^Ctrl;
                          .stViciSerial.stComOut.Ctrl := TIID^MAIN (EtherCAT)^M3 Selector C Serial IO (EP6002-0002)^COM RxPDO-Map Outputs Channel 2^Ctrl;
                          .stShaker01.q_xPwrDO := TIIB[M3 Selector C Digital IO (EP2338-1001)]^Channel 9^Output;
                          .stShaker02.q_xPwrDO := TIIB[M3 Selector C Digital IO (EP2338-1001)]^Channel 10^Output;
                          .stShaker03.q_xPwrDO := TIIB[M3 Selector C Digital IO (EP2338-1001)]^Channel 11^Output;
                          .stShaker04.q_xPwrDO := TIIB[M3 Selector C Digital IO (EP2338-1001)]^Channel 12^Output;
                          .stBaseIO.i_SyncUnitWC := TIID^MAIN (EtherCAT)^M3 Selector C (EP1111)^WcState^WcState
'}
M3SelectorC : FB_SelectorM3;

{attribute 'pytmc' := 'pv: ICL:SDS:SEL:D'}
{attribute 'TcLinkTo' := '.stSensSerial.stComIn.Status := TIIB[M3 Selector D Serial IO (EP6002-0002)]^COM TxPDO-Map Inputs Channel 1^Status;
                          .stViciSerial.stComIn.Status := TIIB[M3 Selector D Serial IO (EP6002-0002)]^COM TxPDO-Map Inputs Channel 2^Status;
                          .stSensSerial.stComOut.Ctrl := TIID^MAIN (EtherCAT)^M3 Selector D Serial IO (EP6002-0002)^COM RxPDO-Map Outputs Channel 1^Ctrl;
                          .stViciSerial.stComOut.Ctrl := TIID^MAIN (EtherCAT)^M3 Selector D Serial IO (EP6002-0002)^COM RxPDO-Map Outputs Channel 2^Ctrl;
                          .stShaker01.q_xPwrDO := TIIB[M3 Selector D Digital IO (EP2338-1001)]^Channel 9^Output;
                          .stShaker02.q_xPwrDO := TIIB[M3 Selector D Digital IO (EP2338-1001)]^Channel 10^Output;
                          .stShaker03.q_xPwrDO := TIIB[M3 Selector D Digital IO (EP2338-1001)]^Channel 11^Output;
                          .stShaker04.q_xPwrDO := TIIB[M3 Selector D Digital IO (EP2338-1001)]^Channel 12^Output;
                          .stBaseIO.i_SyncUnitWC := TIID^MAIN (EtherCAT)^M3 Selector D (EP1111)^WcState^WcState
'}
M3SelectorD : FB_SelectorM3;

{attribute 'pytmc' := 'pv: ICL:SDS:PCM:A'}
{attribute 'TcLinkTo' := '.stPropAir1.i_iPressRB := TIID^MAIN (EtherCAT)^PCM A (EP4374-0002)^AI Inputs Channel 1^Value;
                          .stPropAir2.i_iPressRB := TIID^MAIN (EtherCAT)^PCM A (EP4374-0002)^AI Inputs Channel 2^Value;
                          .stPropAir1.q_iPressCt := TIID^MAIN (EtherCAT)^PCM A (EP4374-0002)^AO Outputs Channel 3^Analog output;
                          .stPropAir2.q_iPressCt := TIID^MAIN (EtherCAT)^PCM A (EP4374-0002)^AO Outputs Channel 4^Analog output;
                          .stSerial1.stComIn.Status := TIID^MAIN (EtherCAT)^PCM A (EP6002-0002)^COM TxPDO-Map Inputs Channel 1^Status;
                          .stSerial2.stComIn.Status := TIID^MAIN (EtherCAT)^PCM A (EP6002-0002)^COM TxPDO-Map Inputs Channel 2^Status;
                          .stSerial1.stComOut.Ctrl := TIID^MAIN (EtherCAT)^PCM A (EP6002-0002)^COM RxPDO-Map Outputs Channel 1^Ctrl;
                          .stSerial2.stComOut.Ctrl := TIID^MAIN (EtherCAT)^PCM A (EP6002-0002)^COM RxPDO-Map Outputs Channel 2^Ctrl;
                          .stBaseIO.i_SyncUnitWC := TIID^MAIN (EtherCAT)^PCM A (EP1111)^WcState^WcState;
'}
PCMA : FB_PressureControlModule;

{attribute 'pytmc' := 'pv: ICL:SDS:PCM:B'}
{attribute 'TcLinkTo' := '.stPropAir1.i_iPressRB := TIID^MAIN (EtherCAT)^PCM B (EP4374-0002)^AI Inputs Channel 1^Value;
                          .stPropAir2.i_iPressRB := TIID^MAIN (EtherCAT)^PCM B (EP4374-0002)^AI Inputs Channel 2^Value;
                          .stPropAir1.q_iPressCt := TIID^MAIN (EtherCAT)^PCM B (EP4374-0002)^AO Outputs Channel 3^Analog output;
                          .stPropAir2.q_iPressCt := TIID^MAIN (EtherCAT)^PCM B (EP4374-0002)^AO Outputs Channel 4^Analog output;
                          .stSerial1.stComIn.Status := TIID^MAIN (EtherCAT)^PCM B (EP6002-0002)^COM TxPDO-Map Inputs Channel 1^Status;
                          .stSerial2.stComIn.Status := TIID^MAIN (EtherCAT)^PCM B (EP6002-0002)^COM TxPDO-Map Inputs Channel 2^Status;
                          .stSerial1.stComOut.Ctrl := TIID^MAIN (EtherCAT)^PCM B (EP6002-0002)^COM RxPDO-Map Outputs Channel 1^Ctrl;
                          .stSerial2.stComOut.Ctrl := TIID^MAIN (EtherCAT)^PCM B (EP6002-0002)^COM RxPDO-Map Outputs Channel 2^Ctrl;
                          .stBaseIO.i_SyncUnitWC := TIID^MAIN (EtherCAT)^PCM B (EP1111)^WcState^WcState;

'}
PCMB : FB_PressureControlModule;

{attribute 'pytmc' := 'pv: ICL:SDS:PCM:C'}
{attribute 'TcLinkTo' := '.stPropAir1.i_iPressRB := TIID^MAIN (EtherCAT)^PCM C (EP4374-0002)^AI Inputs Channel 1^Value;
                          .stPropAir2.i_iPressRB := TIID^MAIN (EtherCAT)^PCM C (EP4374-0002)^AI Inputs Channel 2^Value;
                          .stPropAir1.q_iPressCt := TIID^MAIN (EtherCAT)^PCM C (EP4374-0002)^AO Outputs Channel 3^Analog output;
                          .stPropAir2.q_iPressCt := TIID^MAIN (EtherCAT)^PCM C (EP4374-0002)^AO Outputs Channel 4^Analog output;
                          .stSerial1.stComIn.Status := TIID^MAIN (EtherCAT)^PCM C (EP6002-0002)^COM TxPDO-Map Inputs Channel 1^Status;
                          .stSerial2.stComIn.Status := TIID^MAIN (EtherCAT)^PCM C (EP6002-0002)^COM TxPDO-Map Inputs Channel 2^Status;
                          .stSerial1.stComOut.Ctrl := TIID^MAIN (EtherCAT)^PCM C (EP6002-0002)^COM RxPDO-Map Outputs Channel 1^Ctrl;
                          .stSerial2.stComOut.Ctrl := TIID^MAIN (EtherCAT)^PCM C (EP6002-0002)^COM RxPDO-Map Outputs Channel 2^Ctrl;
                          .stBaseIO.i_SyncUnitWC := TIID^MAIN (EtherCAT)^PCM C (EP1111)^WcState^WcState;
'}
PCMC : FB_PressureControlModule;

{attribute 'pytmc' := 'pv: ICL:SDS:PCM:D'}
{attribute 'TcLinkTo' := '.stPropAir1.i_iPressRB := TIID^MAIN (EtherCAT)^PCM D (EP4374-0002)^AI Inputs Channel 1^Value;
                          .stPropAir2.i_iPressRB := TIID^MAIN (EtherCAT)^PCM D (EP4374-0002)^AI Inputs Channel 2^Value;
                          .stPropAir1.q_iPressCt := TIID^MAIN (EtherCAT)^PCM D (EP4374-0002)^AO Outputs Channel 3^Analog output;
                          .stPropAir2.q_iPressCt := TIID^MAIN (EtherCAT)^PCM D (EP4374-0002)^AO Outputs Channel 4^Analog output;
                          .stSerial1.stComIn.Status := TIID^MAIN (EtherCAT)^PCM D (EP6002-0002)^COM TxPDO-Map Inputs Channel 1^Status;
                          .stSerial2.stComIn.Status := TIID^MAIN (EtherCAT)^PCM D (EP6002-0002)^COM TxPDO-Map Inputs Channel 2^Status;
                          .stSerial1.stComOut.Ctrl := TIID^MAIN (EtherCAT)^PCM D (EP6002-0002)^COM RxPDO-Map Outputs Channel 1^Ctrl;
                          .stSerial2.stComOut.Ctrl := TIID^MAIN (EtherCAT)^PCM D (EP6002-0002)^COM RxPDO-Map Outputs Channel 2^Ctrl;
                          .stBaseIO.i_SyncUnitWC := TIID^MAIN (EtherCAT)^PCM D (EP1111)^WcState^WcState;
'}
PCMD : FB_PressureControlModule;

{attribute 'pytmc' := 'pv: ICL:SDS:MAN'}
{attribute 'TcLinkTo' := '.stValve[1].qxDO := TIIB[Gas_Mani_ValveCtrl (EP2338-0001)]^Channel 9^Output;
                          .stValve[1].ixOPN := TIIB[Gas_Mani_ValveRbk (EP2338-0001)]^Channel 1^Input;
                          .stValve[2].qxDO := TIIB[Gas_Mani_ValveCtrl (EP2338-0001)]^Channel 10^Output;
                          .stValve[2].ixOPN := TIIB[Gas_Mani_ValveRbk (EP2338-0001)]^Channel 2^Input;
                          .stValve[3].qxDO := TIIB[Gas_Mani_ValveCtrl (EP2338-0001)]^Channel 11^Output;
                          .stValve[3].ixOPN := TIIB[Gas_Mani_ValveRbk (EP2338-0001)]^Channel 3^Input;
                          .stValve[4].qxDO := TIIB[Gas_Mani_ValveCtrl (EP2338-0001)]^Channel 12^Output;
                          .stValve[4].ixOPN := TIIB[Gas_Mani_ValveRbk (EP2338-0001)]^Channel 4^Input;
                          .stValve[5].qxDO := TIIB[Gas_Mani_ValveCtrl (EP2338-0001)]^Channel 13^Output;
                          .stValve[5].ixOPN := TIIB[Gas_Mani_ValveRbk (EP2338-0001)]^Channel 5^Input;
                          .stValve[6].qxDO := TIIB[Gas_Mani_ValveCtrl (EP2338-0001)]^Channel 14^Output;
                          .stValve[6].ixOPN := TIIB[Gas_Mani_ValveRbk (EP2338-0001)]^Channel 6^Input;
                          .stValve[7].qxDO := TIIB[Gas_Mani_ValveCtrl (EP2338-0001)]^Channel 15^Output;
                          .stValve[7].ixOPN := TIIB[Gas_Mani_ValveRbk (EP2338-0001)]^Channel 7^Input;
                          .stBaseIO.i_SyncUnitWC :=	TIID^MAIN (EtherCAT)^Gas_Mani (EP1111)^WcState^WcState;
'}
GasMan : FB_GasManifold;

{attribute 'pytmc' := 'pv: ICL:SDS:MFM:A'}
{attribute 'TcLinkTo' := '.stMFM.i_rFlow := TIID^MAIN (EtherCAT)^Bronkhorst MFM A^TxPDO Map^fMeasure;
                          .stMFM.q_rSetpoint := TIID^MAIN (EtherCAT)^Bronkhorst MFM A^RxPDO Map^fSetpoint;
'}
BronkhorstA : FB_BronkhorstMFM;

{attribute 'pytmc' := 'pv: ICL:SDS:MFM:B'}
{attribute 'TcLinkTo' := '.stMFM.i_rFlow := TIID^MAIN (EtherCAT)^Bronkhorst MFM B^TxPDO Map^fMeasure;
                          .stMFM.q_rSetpoint := TIID^MAIN (EtherCAT)^Bronkhorst MFM B^RxPDO Map^fSetpoint;
'}
BronkhorstB : FB_BronkhorstMFM;

{attribute 'pytmc' := 'pv: ICL:SDS:MFM:C'}
{attribute 'TcLinkTo' := '.stMFM.i_rFlow := TIID^MAIN (EtherCAT)^Bronkhorst MFM C^TxPDO Map^fMeasure;
                          .stMFM.q_rSetpoint := TIID^MAIN (EtherCAT)^Bronkhorst MFM C^RxPDO Map^fSetpoint;
'}
BronkhorstC : FB_BronkhorstMFM;

{attribute 'pytmc' := 'pv: ICL:SDS:MFM:D'}
{attribute 'TcLinkTo' := '.stMFM.i_rFlow := TIID^MAIN (EtherCAT)^Bronkhorst MFM D^TxPDO Map^fMeasure;
                          .stMFM.q_rSetpoint := TIID^MAIN (EtherCAT)^Bronkhorst MFM D^RxPDO Map^fSetpoint;
'}
BronkhorstD : FB_BronkhorstMFM;

{attribute 'pytmc' := 'pv: ICL:SDS:SPR:A'}
{attribute 'TcLinkTo' := '.q_xDO1 := TIIB[Solenoid Pair A Digital IO (EP2338-0001)]^Channel 9^Output;
                          .q_xDO2 := TIIB[Solenoid Pair A Digital IO (EP2338-0001)]^Channel 10^Output;
'}
SolenoidPairA : FB_SolenoidPair;




END_VAR

// ---- POUs/MAIN.TcPOU
PROGRAM MAIN
VAR

END_VAR

fbSelectorA();

(* Following execution of all the programs, set the first pass false *)
g_xFirstPass := FALSE;

END_PROGRAM
